FUNCTION FC 23 : VOID
TITLE = Bock for actuating several cycled valves
//Erstellung:
//Datum       Bearbeiter                                                   Version
//--------------------------------------------------------------------------------
//14.06.99    A.Kirchgessner(kia)                                         01.00.00
//
//Änderungen:
//Nr. Datum    Bearb Änderung                                       Marke  Version
//--------------------------------------------------------------------------------
//01  16.07.99 kia   Fehlerbeseitigung                                    01.00.01
//02  12.08.99 sra   Fehlerbeseitigung mit Parameteränderung              01.01.00
//03  19.10.99 sra   Anpassung an neue Struktur                           01.02.00
//04  10.07.00 sra   Fehlerbeseitigung Taktgenerierung                    01.02.01
//05  10.07.00 sra   Änderung in Eingangsparameter                        01.03.00
//06  19.09.00 sra   komplette Überarbeitung / neue Struktur              02.00.00
//07  18.01.01 gea   Erweiterung auf 10 Ventile / neue Struktur           02.01.00
//08  27.03.02 sra   Meldung "Ventil in Betrieb" auch im Handmode   (008) 02.01.01
//09  04.02.03 kal   Fehlerbeseitigung Dauertakt                    (009) 02.01.02
//10  31.10.05 sra   Ansteuerung Handbedienung im Automode rücksetz.
//                   Handbedienung zentral sperren                  (010) 02.02.00
//11  18.02.09 kmj   Objektststatus für OP ergänzt                  (011) 02.03.00
//12  20.03.09 kal   Objektststatus für OP ergänzt (überarbeitet)   (012) 02.03.01
//13  24.04.09 gea   Handmode zurücksetzen wenn Handmode gesperrt   (013) 02.03.02
//14  05.12.13 sra   "Anlage ein" eingefügt (Not-Aus-Konzept)       (014) 02.04.00
//15  14.11.14 bhl   Anzeige "#io_Ventil_in_Betrieb" im Handmode    (015) 02.04.01
//16  11.08.15 sra   "#io_Ventil_in_Betrieb" nur wenn "Anlage ein"  (016) 02.04.02
//________________________________________________________________________________
//Eingesetzte Bausteine:
//
//FC2 : Version 01.01.XX
//________________________________________________________________________________
//Funktion:
//
//Der Baustein taktet die einzelnen Ventile der Reihe nach durch (Anzahl der 
//Ventile max. 10 Stück). 
//
//Die Ausgänge werden nur angesteuert wenn der Eingang "in_Anlage_ein" = true
//ist. Diese Funktion ist vorhanden, um bei einem Not-Halt die Anlage vor 
//unkontrolliertem Einschalten zu schützen. 
//
//Im Handmode werden die ausgewählten Ventile dauerhaft angesteuert. 
//
AUTHOR : kia
FAMILY : AZO
VERSION : 0.0
VAR_INPUT
  in_Handbedienung_erlaubt : BOOL ;	//1 = manual operation permitted, 0 = manual operation not permitted/locked
  in_Anlage_ein : BOOL ;	//Anlage bzw. Anlagenbereich nach Not-Halt freigegeben
  in_Ansteuerung_Ventil_T1 : BOOL ;	//Actuation of valve position 1 in automatic mode with cycle 1
  in_Ansteuerung_Ventil_T2 : BOOL ;	//Actuation of valve position 1 in automatic mode with cycle 2
END_VAR
VAR_IN_OUT
  io_Ausgang_Ventil_1 : BOOL ;	//Output 1. Valve
  io_Ausgang_Ventil_2 : BOOL ;	//Output 2. Valve
  io_Ausgang_Ventil_3 : BOOL ;	//Output 3. Valve
  io_Ausgang_Ventil_4 : BOOL ;	//Output 4. Valve
  io_Ausgang_Ventil_5 : BOOL ;	//Output 5. Valve
  io_Ausgang_Ventil_6 : BOOL ;	//Output 6. Valve
  io_Ausgang_Ventil_7 : BOOL ;	//Output 7. Valve
  io_Ausgang_Ventil_8 : BOOL ;	//Output 8. Valve
  io_Ausgang_Ventil_9 : BOOL ;	//Output 9. Valve
  io_Ausgang_Ventil_10 : BOOL ;	//Output 10. Valve
  io_Ventil_in_Betrieb : BOOL ;	//Signal "valve in operation" (actuated)
  io_Ventilstruktur : ANY ;	//ANY pointer of valve structure
END_VAR
VAR_TEMP
  Ventilansteuerung : BOOL ;	//Freigabe ein Ventil anzusteuern
  Freigabe_Takt : BOOL ;	//Cycle enable
  Rueckmeldung : BOOL ;	//wenn eines der Ventil agesteuert ist --> 1-Signal
  Start_mit_Impuls : BOOL ;
  Taktanzahl_erreicht : BOOL ;
  Dauertakt : BOOL ;	//Continuous cycle
  positive_Flanke : BOOL ;
  Hilfs_Anzahl_Takte : INT ;	//Sollvorgabe für FC2
  Aktuelles_Ventil : INT ;	//aktuelles Ventil
  Hilfswort_1 : INT ;
  Impulszeit_Takt : REAL ;
  Pausezeit_Takt : REAL ;
  Zeitzaehler : REAL ;
  Taktzaehler : INT ;
  Objektstatus : INT ;
END_VAR
BEGIN
NETWORK
TITLE = Anfangs-DW der Struktur aus ANY-Zeiger auslesen
      L     P##io_Ventilstruktur;
      LAR2;
      L     D [AR2,P#6.0];
      LAR2;	//Pointer auf Structuranfang
NETWORK
TITLE = Umschaltung Hand-/Automatikmode 
      A     DIX [AR2,P#3.6];	// Handmode von Farbgrafik (Struktur)
      AN    DIX [AR2,P#5.1];	// Handmode gesperrt (Struktur)
      AN    M 0.0;	// Handbedienung zentral sperren (010)
      S     DIX [AR2,P#3.5];	// Handmode zu Farbgrafik (Struktur)
      ON    DIX [AR2,P#3.6];	// Handmode von Farbgrafik (Struktur)
      ON    #in_Handbedienung_erlaubt;
      O     M 0.0;	// Handbedienung zentral sperren (010)
      O     DIX [AR2,P#5.1];	// Handmode gesperrt (Struktur) (013)
      R     DIX [AR2,P#3.5];	// Handmode zu Farbgrafik (Struktur)
      R     DIX [AR2,P#3.6];	// Handmode von Farbgrafik (Struktur) (010)
NETWORK
TITLE = Ansteuerung Handmode zurücksetzen
//(010) 
      AN    DIX [AR2,P#3.5];	// Handmode zu Farbgrafik (Struktur)
      R     DIX [AR2,P#3.7];	// Ansteuerung des 1. Ventils im Handmode von Farbgrafik (Struktur)
      R     DIX [AR2,P#4.0];	// Ansteuerung des 2. Ventils im Handmode von Farbgrafik (Struktur)
      R     DIX [AR2,P#4.1];	// Ansteuerung des 3. Ventils im Handmode von Farbgrafik (Struktur)
      R     DIX [AR2,P#4.2];	// Ansteuerung des 4. Ventils im Handmode von Farbgrafik (Struktur)
      R     DIX [AR2,P#4.3];	// Ansteuerung des 5. Ventils im Handmode von Farbgrafik (Struktur)
      R     DIX [AR2,P#4.4];	// Ansteuerung des 6. Ventils im Handmode von Farbgrafik (Struktur)
      R     DIX [AR2,P#4.5];	// Ansteuerung des 7. Ventils im Handmode von Farbgrafik (Struktur)
      R     DIX [AR2,P#4.6];	// Ansteuerung des 8. Ventils im Handmode von Farbgrafik (Struktur)
      R     DIX [AR2,P#4.7];	// Ansteuerung des 9. Ventils im Handmode von Farbgrafik (Struktur)
      R     DIX [AR2,P#5.0];	// Ansteuerung des 10. Ventils im Handmode von Farbgrafik (Struktur)
NETWORK
TITLE = Rueckmeldung Ventile + Ventilansteuerung
      O     #io_Ausgang_Ventil_1;
      O     #io_Ausgang_Ventil_2;
      O     #io_Ausgang_Ventil_3;
      O     #io_Ausgang_Ventil_4;
      O     #io_Ausgang_Ventil_5;
      O     #io_Ausgang_Ventil_6;
      O     #io_Ausgang_Ventil_7;
      O     #io_Ausgang_Ventil_8;
      O     #io_Ausgang_Ventil_9;
      O     #io_Ausgang_Ventil_10;
      =     #Rueckmeldung;
      =     #Ventilansteuerung;
NETWORK
TITLE = Daten für Takt in temporäre Variablen laden
//(009) komplettes Netzwerk gelöscht.
//Dauertakt nur, wenn Bit in Struktur = TRUE 
//Anzahl Takte ist egal!!!
      A     DIX [AR2,P#5.2];	// Start mit Impuls (Struktur)
      =     #Start_mit_Impuls;
      A     DIX [AR2,P#5.3];	// Taktanzahl erreicht (Struktur)
      =     #Taktanzahl_erreicht;
      A     DIX [AR2,P#5.4];	// Dauertakt (Struktur)
      =     #Dauertakt;
      L     DID [AR2,P#22.0];	// Impuls-/Pausezähler (Struktur)
      T     #Zeitzaehler;
      L     DIW [AR2,P#28.0];	// Taktzähler (Struktur)
      T     #Taktzaehler;
NETWORK
TITLE = Sollanzahl Takte
      AN    #Dauertakt;
      JC    ST_1;
      L     DIW [AR2,P#30.0];	// Anzahl Ventile (Struktur)
      T     #Hilfs_Anzahl_Takte;
ST_1: NOP   0;
      A     #Dauertakt;
      JC    ST_2;
      L     DIW [AR2,P#26.0];	// Sollanzahl Takte (Struktur)
      T     #Hilfs_Anzahl_Takte;
ST_2: NOP   0;
NETWORK
TITLE = Freigabe Takt
      A     #in_Anlage_ein;	// (014)
      A(;	// (014)
      O     #in_Ansteuerung_Ventil_T1;
      O     #in_Ansteuerung_Ventil_T2;
      );	// (014)
      =     #Freigabe_Takt;
NETWORK
TITLE = Takt umkopieren
      L     DID [AR2,P#6.0];	// Impulszeit Befüllung (Struktur)
      T     #Impulszeit_Takt;
      L     DID [AR2,P#10.0];	// Pausezeit Befüllung (Struktur)
      T     #Pausezeit_Takt;
      A     #in_Ansteuerung_Ventil_T1;
      JC    E_Tk;
      L     DID [AR2,P#14.0];	// Impulszeit Entleerung (Struktur)
      T     #Impulszeit_Takt;
      L     DID [AR2,P#18.0];	// Pausezeit Entleerung (Struktur)
      T     #Pausezeit_Takt;
E_Tk: NOP   0;
NETWORK
TITLE = Takt generieren
      CALL  FC 2 (
           in_Freigabe              := #Freigabe_Takt,
           in_Rueckmeldung          := #Rueckmeldung,
           in_Start_mit_Impuls      := #Start_mit_Impuls,
           in_Dauertakt             := #Dauertakt,
           in_Impuls                := M 1.7,
           in_Impulszeit_in_100ms   := MW 6,
           in_Impulszeit            := #Impulszeit_Takt,
           in_Pausezeit             := #Pausezeit_Takt,
           in_Sollanzahl_Takte      := #Hilfs_Anzahl_Takte,
           io_Taktausgang           := #Ventilansteuerung,
           io_Taktanzahl_erreicht   := #Taktanzahl_erreicht,
           io_Zeitzaehler           := #Zeitzaehler,
           io_Taktzaehler           := #Taktzaehler);
NETWORK
TITLE = aktuelles Ventil
      L     #Taktzaehler;
      L     DIW [AR2,P#30.0];	// Anzahl Ventile (Struktur)
      /I;
      T     #Hilfswort_1;
      L     #Hilfswort_1;
      L     DIW [AR2,P#30.0];	// Anzahl Ventile (Struktur)
      *I;
      L     -1;
      *I;
      L     #Taktzaehler;
      +I;
      L     1;
      +I;
      T     #Aktuelles_Ventil;
NETWORK
TITLE = aktuelles Ventil prüfen
      A(;
      L     #Aktuelles_Ventil;
      L     1;
      >=I;
      );
      A(;
      L     #Aktuelles_Ventil;
      L     DIW [AR2,P#30.0];	// Anzahl Ventile (Struktur)
      <=I;
      );
      JC    M1;
      L     1;
      T     #Aktuelles_Ventil;
M1:   NOP   0;
NETWORK
TITLE = Ansteuerung Ventil 1
      A     #in_Anlage_ein;	// (014)
      A(;	// (014)
      A(;
      L     #Aktuelles_Ventil;
      L     1;
      ==I;
      );
      A(;	// Automatikmode
      AN    DIX [AR2,P#3.5];	// Handmode zu Farbgrafik (Struktur)
      A     #Ventilansteuerung;
      AN    #Taktanzahl_erreicht;
      );
      O;	// Handmode 
      A     DIX [AR2,P#3.5];	// Handmode zu Farbgrafik (Struktur)
      A     DIX [AR2,P#3.7];	// Ansteuerung des 1. Ventils im Handmode von Farbgrafik (Struktur)
      );	// (014)
      =     #io_Ausgang_Ventil_1;
NETWORK
TITLE = Ansteuerung Ventil 2
      A     #in_Anlage_ein;	// (014)
      A(;	// (014)
      A(;
      L     #Aktuelles_Ventil;
      L     2;
      ==I;
      );
      A(;	// Automatikmode
      AN    DIX [AR2,P#3.5];	// Handmode zu Farbgrafik (Struktur)
      A     #Ventilansteuerung;
      AN    #Taktanzahl_erreicht;
      );
      O;	// Handmode 
      A     DIX [AR2,P#3.5];	// Handmode zu Farbgrafik (Struktur)
      A     DIX [AR2,P#4.0];	// Ansteuerung des 2. Ventils im Handmode von Farbgrafik (Struktur)
      );	// (014)
      =     #io_Ausgang_Ventil_2;
NETWORK
TITLE = Ansteuerung Ventil 3
      A     #in_Anlage_ein;	// (014)
      A(;	// (014)
      A(;
      L     #Aktuelles_Ventil;
      L     3;
      ==I;
      );
      A(;	// Automatikmode
      AN    DIX [AR2,P#3.5];	// Handmode zu Farbgrafik (Struktur)
      A     #Ventilansteuerung;
      AN    #Taktanzahl_erreicht;
      );
      O;	// Handmode 
      A     DIX [AR2,P#3.5];	// Handmode zu Farbgrafik (Struktur)
      A     DIX [AR2,P#4.1];	// Ansteuerung des 3. Ventils im Handmode von Farbgrafik (Struktur)
      );	// (014)
      =     #io_Ausgang_Ventil_3;
NETWORK
TITLE = Ansteuerung Ventil 4
      A     #in_Anlage_ein;	// (014)
      A(;	// (014)
      A(;
      L     #Aktuelles_Ventil;
      L     4;
      ==I;
      );
      A(;	// Automatikmode
      AN    DIX [AR2,P#3.5];	// Handmode zu Farbgrafik (Struktur)
      A     #Ventilansteuerung;
      AN    #Taktanzahl_erreicht;
      );
      O;	// Handmode 
      A     DIX [AR2,P#3.5];	// Handmode zu Farbgrafik (Struktur)
      A     DIX [AR2,P#4.2];	// Ansteuerung des 4. Ventils im Handmode von Farbgrafik (Struktur)
      );	// (014)
      =     #io_Ausgang_Ventil_4;
NETWORK
TITLE = Ansteuerung Ventil 5
      A     #in_Anlage_ein;	// (014)
      A(;	// (014)
      A(;
      L     #Aktuelles_Ventil;
      L     5;
      ==I;
      );
      A(;	// Automatikmode
      AN    DIX [AR2,P#3.5];	// Handmode zu Farbgrafik (Struktur)
      A     #Ventilansteuerung;
      AN    #Taktanzahl_erreicht;
      );
      O;	// Handmode 
      A     DIX [AR2,P#3.5];	// Handmode zu Farbgrafik (Struktur)
      A     DIX [AR2,P#4.3];	// Ansteuerung des 5. Ventils im Handmode von Farbgrafik (Struktur)
      );	// (014)
      =     #io_Ausgang_Ventil_5;
NETWORK
TITLE = Ansteuerung Ventil 6
      A     #in_Anlage_ein;	// (014)
      A(;	// (014)
      A(;
      L     #Aktuelles_Ventil;
      L     6;
      ==I;
      );
      A(;	// Automatikmode
      AN    DIX [AR2,P#3.5];	// Handmode zu Farbgrafik (Struktur)
      A     #Ventilansteuerung;
      AN    #Taktanzahl_erreicht;
      );
      O;	// Handmode 
      A     DIX [AR2,P#3.5];	// Handmode zu Farbgrafik (Struktur)
      A     DIX [AR2,P#4.4];	// Ansteuerung des 6. Ventils im Handmode von Farbgrafik (Struktur)
      );	// (014)
      =     #io_Ausgang_Ventil_6;
NETWORK
TITLE = Ansteuerung Ventil 7
      A     #in_Anlage_ein;	// (014)
      A(;	// (014)
      A(;
      L     #Aktuelles_Ventil;
      L     7;
      ==I;
      );
      A(;	// Automatikmode
      AN    DIX [AR2,P#3.5];	// Handmode zu Farbgrafik (Struktur)
      A     #Ventilansteuerung;
      AN    #Taktanzahl_erreicht;
      );
      O;	// Handmode 
      A     DIX [AR2,P#3.5];	// Handmode zu Farbgrafik (Struktur)
      A     DIX [AR2,P#4.5];	// Ansteuerung des 7. Ventils im Handmode von Farbgrafik (Struktur)
      );	// (014)
      =     #io_Ausgang_Ventil_7;
NETWORK
TITLE = Ansteuerung Ventil 8
      A     #in_Anlage_ein;	// (014)
      A(;	// (014)
      A(;
      L     #Aktuelles_Ventil;
      L     8;
      ==I;
      );
      A(;	// Automatikmode
      AN    DIX [AR2,P#3.5];	// Handmode zu Farbgrafik (Struktur)
      A     #Ventilansteuerung;
      AN    #Taktanzahl_erreicht;
      );
      O;	// Handmode 
      A     DIX [AR2,P#3.5];	// Handmode zu Farbgrafik (Struktur)
      A     DIX [AR2,P#4.6];	// Ansteuerung des 8. Ventils im Handmode von Farbgrafik (Struktur)
      );	// (014)
      =     #io_Ausgang_Ventil_8;
NETWORK
TITLE = Ansteuerung Ventil 9
      A     #in_Anlage_ein;	// (014)
      A(;	// (014)
      A(;
      L     #Aktuelles_Ventil;
      L     9;
      ==I;
      );
      A(;	// Automatikmode
      AN    DIX [AR2,P#3.5];	// Handmode zu Farbgrafik (Struktur)
      A     #Ventilansteuerung;
      AN    #Taktanzahl_erreicht;
      );
      O;	// Handmode 
      A     DIX [AR2,P#3.5];	// Handmode zu Farbgrafik (Struktur)
      A     DIX [AR2,P#4.7];	// Ansteuerung des 9. Ventils im Handmode von Farbgrafik (Struktur)
      );	// (014)
      =     #io_Ausgang_Ventil_9;
NETWORK
TITLE = Ansteuerung Ventil 10
      A     #in_Anlage_ein;	// (014)
      A(;	// (014)
      A(;
      L     #Aktuelles_Ventil;
      L     10;
      ==I;
      );
      A(;	// Automatikmode
      AN    DIX [AR2,P#3.5];	// Handmode zu Farbgrafik (Struktur)
      A     #Ventilansteuerung;
      AN    #Taktanzahl_erreicht;
      );
      O;	// Handmode 
      A     DIX [AR2,P#3.5];	// Handmode zu Farbgrafik (Struktur)
      A     DIX [AR2,P#5.0];	// Ansteuerung des 10. Ventils im Handmode von Farbgrafik (Struktur)
      );	// (014)
      =     #io_Ausgang_Ventil_10;
NETWORK
TITLE = Ausgang Betrieb
      AN    DIX [AR2,P#3.5];	// (015) Handmode zu Farbgrafik (Struktur)
      A     #in_Anlage_ein;	// (016)
      A(;
      O     #in_Ansteuerung_Ventil_T1;
      O     #in_Ansteuerung_Ventil_T2;	// (008)
      );
      A     #Dauertakt;
      O;
      AN    DIX [AR2,P#3.5];	// (015) Handmode zu Farbgrafik (Struktur)
      A     #in_Anlage_ein;	// (016)
      A(;
      O     #in_Ansteuerung_Ventil_T1;
      O     #in_Ansteuerung_Ventil_T2;
      );
      AN    #Dauertakt;
      AN    #Taktanzahl_erreicht;
      O;
      A     DIX [AR2,P#3.5];	// Handmode zu Farbgrafik (Struktur)
      A     #in_Anlage_ein;	// (016)
      A(;
      O     #io_Ausgang_Ventil_1;	// (008)
      O     #io_Ausgang_Ventil_2;	// (008)
      O     #io_Ausgang_Ventil_3;	// (008)
      O     #io_Ausgang_Ventil_4;	// (008)
      O     #io_Ausgang_Ventil_5;	// (008)
      O     #io_Ausgang_Ventil_6;	// (008)
      O     #io_Ausgang_Ventil_7;	// (008)
      O     #io_Ausgang_Ventil_8;	// (008)
      O     #io_Ausgang_Ventil_9;	// (008)
      O     #io_Ausgang_Ventil_10;	// (008)
      );
      =     #io_Ventil_in_Betrieb;
NETWORK
TITLE = Flankenauswertung Ausgang Ventil für Schalthäufigkeitzähler
//Es wird die Schalthäufigkeit der Ventile gezählt !  
      O     #io_Ausgang_Ventil_1;
      O     #io_Ausgang_Ventil_2;
      O     #io_Ausgang_Ventil_3;
      O     #io_Ausgang_Ventil_4;
      O     #io_Ausgang_Ventil_5;
      O     #io_Ausgang_Ventil_6;
      O     #io_Ausgang_Ventil_7;
      O     #io_Ausgang_Ventil_8;
      O     #io_Ausgang_Ventil_9;
      O     #io_Ausgang_Ventil_10;
      FP    DIX [AR2,P#32.3];	// Flankenmerker Ausgang (Struktur)
      =     #positive_Flanke;
NETWORK
TITLE = Schalthäufigkeitzähler
      ON    DIX [AR2,P#0.3];	// Kennung Schalthäufigkeitzähler ein (Struktur)
      ON    #positive_Flanke;
      JC    ESHZ;
      L     1.000000e+00;
      L     DID [AR2,P#34.0];	// Schalthäufigkeitzähler (Struktur)
      +R;
      T     DID [AR2,P#34.0];	// Schalthäufigkeitzähler (Struktur)
ESHZ: NOP   0;
NETWORK
TITLE = Schalthäufigkeitzähler zurücksetzten
      AN    DIX [AR2,P#32.0];	// Reset Schalthäufigkeitzähler (Struktur)
      JC    E_RS;
      L     0.000000e+00;
      T     DID [AR2,P#34.0];	// Schalthäufigkeitzähler (Struktur)
      CLR;
      =     DIX [AR2,P#32.0];	// Reset Schalthäufigkeitzähler (Struktur)
E_RS: NOP   0;
NETWORK
TITLE = Warnmeldung Schalthäufigkeitzähler erzeugen
      A(;
      L     DID [AR2,P#34.0];	// Schalthäufigkeitzähler (Struktur)
      L     DID [AR2,P#38.0];	// Sollwert Warnung (Struktur)
      >R;
      );
      A(;
      L     DID [AR2,P#38.0];	// Sollwert Warnung (Struktur)
      L     0.000000e+00;
      <>R;
      );
      =     DIX [AR2,P#32.1];	// Warnmeldung Schalthäufigkeitzähler (Struktur)
NETWORK
TITLE = Alarmmeldung Schalthäufigkeitzähler erzeugen
      A(;
      L     DID [AR2,P#34.0];	// Schalthäufigkeitzähler (Struktur)
      L     DID [AR2,P#42.0];	// Sollwert Alarm (Struktur)
      >R;
      );
      A(;
      L     DID [AR2,P#42.0];	// Sollwert Alarm (Struktur)
      L     0.000000e+00;
      <>R;
      );
      =     DIX [AR2,P#32.2];	// Warnmeldung Schalthäufigkeitzähler (Struktur)
NETWORK
TITLE = Objektstatus für Visualisation OP (011)(012)
//Stati:
//-------
//1 = kein Ventil angesteuert ==> Farbvorschlag weiß
//5 = ein ventil in Betrieb ==> Farbvorschlag grün
//
// 1 = nicht in Betrieb, keine Störung ==> Farbvorschlag grau
      L     1;
      AN    #io_Ventil_in_Betrieb;
      JC    disp;
// 5 = angesteuert, nicht in Betrieb, keine Störung ==> Farbvorschlag grün
      L     5;
      A     #io_Ventil_in_Betrieb;
      JC    disp;
      L     0;
disp: T     #Objektstatus;
NETWORK
TITLE = Daten in Struktur speichern
      A     #in_Anlage_ein;	// (014)
      =     DIX [AR2,P#5.5];	// (014) Anlage ein (Struktur)
      A     #io_Ausgang_Ventil_1;
      =     DIX [AR2,P#2.0];	// Ausgang Ventil 1 (Struktur)
      A     #io_Ausgang_Ventil_2;
      =     DIX [AR2,P#2.1];	// Ausgang Ventil 2 (Struktur)
      A     #io_Ausgang_Ventil_3;
      =     DIX [AR2,P#2.2];	// Ausgang Ventil 3 (Struktur)
      A     #io_Ausgang_Ventil_4;
      =     DIX [AR2,P#2.3];	// Ausgang Ventil 4 (Struktur)
      A     #io_Ausgang_Ventil_5;
      =     DIX [AR2,P#2.4];	// Ausgang Ventil 5 (Struktur)
      A     #io_Ausgang_Ventil_6;
      =     DIX [AR2,P#2.5];	// Ausgang Ventil 6 (Struktur)
      A     #io_Ausgang_Ventil_7;
      =     DIX [AR2,P#2.6];	// Ausgang Ventil 7 (Struktur)
      A     #io_Ausgang_Ventil_8;
      =     DIX [AR2,P#2.7];	// Ausgang Ventil 8 (Struktur)
      A     #io_Ausgang_Ventil_9;
      =     DIX [AR2,P#3.0];	// Ausgang Ventil 9 (Struktur)
      A     #io_Ausgang_Ventil_10;
      =     DIX [AR2,P#3.1];	// Ausgang Ventil 10 (Struktur)
      A     #io_Ventil_in_Betrieb;
      =     DIX [AR2,P#3.4];	// Ventil in Betrieb (Struktur)
      A     #Taktanzahl_erreicht;
      =     DIX [AR2,P#5.3];	// Taktanzahl erreicht (Struktur)
      L     #Zeitzaehler;
      T     DID [AR2,P#22.0];	// Impuls-/Pausezähler (Struktur)
      L     #Taktzaehler;
      T     DIW [AR2,P#28.0];	// Taktzähler (Struktur)
      L     #Objektstatus;	// (011)
      T     DIW [AR2,P#48.0];	// #Objektstatus  (Struktur)   // (011)
END_FUNCTION

FUNCTION FC 24 : VOID
TITLE = Block for debouncing and fault monitoring of a binary input
//Building:
//Date         Editor                                                     Version
//--------------------------------------------------------------------------------
//22.09.99     (jm)                                                       01.00.00
//
//Modifications:
//No. Date     Edit  Description                                    Index Version
//--------------------------------------------------------------------------------
//01  29.09.00 sra   komplette Überarbeitung / neue Struktur        ()    02.00.00
//02  16.06.05 sra   Änderung INC 1 -> + 1                         (002)  02.00.01
//03  04.09.06 sra   Änderung Störungsquittierung                  (003)  02.01.00
//04  08.07.10 jm    Störzeit 0 möglich                            (004)  02.01.01
//05  06.06.16 kal/sra komplette Überarbeitung (wie TIA-Portal)     ()    03.00.00
//06  12.06.16 sra   Änderung Signal "Eingang verarbeitet"         (006)  03.01.00
//07  13.12.17 gea   Objektstatus betätig/störung (neu)            (007)  03.02.00
//                   Objektstatus nicht betätig/störung (neu)
//                   Eingang verarbeitet bei Störung ausgeben
//08  26.01.18 gea   Objektstatus Fehlerbeseitigung                (008)  03.02.01
//
//________________________________________________________________________________
//Functional description:
//
//The Binary Input Object includes the following functions
//- The input can be turned (0 = input is active) -> configuration value
//- Depending on the Parameter "in_fault_state", it is possible to select whether
//  log. 0 or log. 1 will represent the fault.
//- The input signal can be debounced in both directions with a seperate time
//  -> Real values in structure
//- The input signal can be counted -> value in structure -> configuration value
//
//The main application for the function are level indicators.
//
AUTHOR : jm
VERSION : 3.2
VAR_INPUT
  in_Handbedienung_erlaubt : BOOL ;
  in_Anlage_ein : BOOL ;
  in_Eingang : BOOL ;
  in_Eingang_drehen : BOOL ;
  in_Eingang_entprellen : BOOL ;
  in_Stoerauswertung_aktiv : BOOL ;
  in_Quitt_Stoerung_noetig : BOOL ;
  in_Stoer_Zustand : BOOL ;
  in_Quitt_Stoerung : BOOL ;
END_VAR
VAR_IN_OUT
  io_Eingang_verarbeitet : BOOL ;
  io_Stoerung : BOOL ;
  io_Struktur : ANY ;
END_VAR
VAR_TEMP
  Eingang_nach_Drehung : BOOL ;
  Eingang_nach_Entprellung : BOOL ;
  Diskrepanz : BOOL ;
  Freigabe_Entprellung_HIG : BOOL ;
  Ausgang_Entprellung_HIGH : BOOL ;
  Freigabe_Entprellung_LOW : BOOL ;
  Ausgang_Entprellung_LOW : BOOL ;
  positive_Flanke : BOOL ;
  Objektstatus : INT ;
  Temp_DB : INT ;
  Sollzeit_Entprellung_HIG : REAL ;
  Istzeit_Entprellung_HIGH : REAL ;
  Sollzeit_Entprellung_LOW : REAL ;
  Istzeit_entprellung_LOW : REAL ;
END_VAR
BEGIN
NETWORK
TITLE = Anfangs-DW der Struktur aus ANY-Zeiger auslesen
      L     P##io_Struktur;
      LAR2;
      L     D [AR2,P#6.0];
      LAR2;
NETWORK
TITLE = Daten aus Struktur lesen
      A     DIX [AR2,P#3.4];
      =     #Eingang_nach_Drehung;
      A     DIX [AR2,P#3.5];
      =     #Eingang_nach_Entprellung;
      A     DIX [AR2,P#3.6];
      =     #Ausgang_Entprellung_HIGH;
      A     DIX [AR2,P#3.7];
      =     #Ausgang_Entprellung_LOW;
      L     DID [AR2,P#8.0];
      T     #Sollzeit_Entprellung_HIG;
      L     DID [AR2,P#12.0];
      T     #Istzeit_Entprellung_HIGH;
      L     DID [AR2,P#16.0];
      T     #Sollzeit_Entprellung_LOW;
      L     DID [AR2,P#20.0];
      T     #Istzeit_entprellung_LOW;
NETWORK
TITLE = Eingang ggf. drehen
      A     #in_Eingang;
      AN    #in_Eingang_drehen;
      O;
      AN    #in_Eingang;
      A     #in_Eingang_drehen;
      =     #Eingang_nach_Drehung;
NETWORK
TITLE = Umschaltung Hand-/Automatikmode 
      A     DIX [AR2,P#2.7];	// Handmode von Farbgrafik (Struktur)
      AN    DIX [AR2,P#3.1];	// Handmode gesperrt (Struktur)
      AN    M 0.0;	// Handbedienung zentral sperren 
      S     DIX [AR2,P#2.6];	// Handmode zu Farbgrafik (Struktur)
      ON    DIX [AR2,P#2.7];	// Handmode von Farbgrafik (Struktur)
      ON    #in_Handbedienung_erlaubt;
      O     M 0.0;	// Handbedienung zentral sperren 
      O     DIX [AR2,P#3.1];	// Handmode gesperrt (Struktur)
      R     DIX [AR2,P#2.6];	// Handmode zu Farbgrafik (Struktur)
      R     DIX [AR2,P#2.7];	// Handmode von Farbgrafik (Struktur)
NETWORK
TITLE = Handzustand im Automatikmode speichern
      AN    DIX [AR2,P#2.6];	// Handmode zu Farbgrafik (Struktur)
      JCN   SAM;
      A     #Eingang_nach_Drehung;
      AN    #in_Eingang_drehen;
      =     DIX [AR2,P#3.0];	// Zustand Handmode (Struktur)
      AN    #Eingang_nach_Drehung;
      A     #in_Eingang_drehen;
      =     DIX [AR2,P#3.0];	// Zustand Handmode (Struktur)
SAM:  NOP   0;
NETWORK
TITLE = Zustand nach Drehung im Handmode überschreiben
      A     DIX [AR2,P#2.6];	// Handmode zu Farbgrafik (Struktur)
      JCN   SHM;
      A     DIX [AR2,P#3.0];	// Zustand Handmode (Struktur)
      =     #Eingang_nach_Drehung;
SHM:  NOP   0;
NETWORK
TITLE = Diskrepanz feststellen
// Automode
      AN    DIX [AR2,P#2.6];	// Handmode zu Farbgrafik (Struktur)
      A     #in_Stoerauswertung_aktiv;
      AN    #in_Eingang;	//Störung = log. 0
      AN    #in_Stoer_Zustand;
      O;
      AN    DIX [AR2,P#2.6];	// Handmode zu Farbgrafik (Struktur)
      A     #in_Stoerauswertung_aktiv;
      A     #in_Eingang;	//Störung = log. 1
      A     #in_Stoer_Zustand;
      O;
// Handmode 
      A     DIX [AR2,P#2.6];	// Handmode zu Farbgrafik (Struktur)
      A     #in_Stoerauswertung_aktiv;
      AN    #Eingang_nach_Drehung;	//Störung = log. 0
      AN    #in_Stoer_Zustand;
      O;
      A     DIX [AR2,P#2.6];	// Handmode zu Farbgrafik (Struktur)
      A     #in_Stoerauswertung_aktiv;
      A     #Eingang_nach_Drehung;	//Störung = log. 1
      A     #in_Stoer_Zustand;
      =     #Diskrepanz;
NETWORK
TITLE = Stoerungszaehler
      A     #in_Quitt_Stoerung_noetig;
      AN    #in_Quitt_Stoerung;
      A     #io_Stoerung;
      O;
      A     #Diskrepanz;
      AN    #in_Quitt_Stoerung;
      O;
      AN    #in_Quitt_Stoerung_noetig;
      A     #Diskrepanz;
      JC    SZ1;
      L     0;	// Wenn keine Diskrepanz dann Zähler löschen
      T     DIW [AR2,P#6.0];	// Istzeit Störung (Struktur)
      JU    ESZ;
// Störungszähler in jeder Sekunde erhöhen
SZ1:  O     #io_Stoerung;
      ON    M 4.5;	// Sekundenimpuls (Standardmerker)
      JC    ESZ;
      L     DIW [AR2,P#6.0];	// Istzeit Störung (Struktur)
      +     1;	// (002)
      T     DIW [AR2,P#6.0];	// Istzeit Störung (Struktur)
ESZ:  NOP   0;
NETWORK
TITLE = Störmeldung ausgeben
      L     DIW [AR2,P#6.0];	// Istzeit Störung (Struktur)
      L     DIW [AR2,P#4.0];	// Sollzeit Störung (Struktur)
      >I;
      =     #io_Stoerung;
NETWORK
TITLE = Stoerung quittieren
      O     #Diskrepanz;	// Stoerung steht noch an
      ON    #io_Stoerung;
      JC    ESQ;
      ON    #in_Quitt_Stoerung_noetig;	// Stoerung muß quittiert werden ?
      JC    SQ1;	// Stoerung muß nicht quittiert werden
      A     #in_Quitt_Stoerung;
SQ1:  R     #io_Stoerung;
ESQ:  NOP   0;
NETWORK
TITLE = Entprellung HIGH
      A     #Eingang_nach_Drehung;
      A     #in_Eingang_entprellen;
      =     #Freigabe_Entprellung_HIG;
      CALL  FC 3 (
           in_Freigabe              := #Freigabe_Entprellung_HIG,
           in_Reset                 := M 0.3,
           in_Impuls                := M 1.7,
           in_Impulszeit_in_100ms   := MW 6,
           in_Verzoegerungsart      := B#16#45,
           in_Verzoegerungszeit     := #Sollzeit_Entprellung_HIG,
           io_Ausgangssignal        := #Ausgang_Entprellung_HIGH,
           io_Zeitzaehler           := #Istzeit_Entprellung_HIGH);
NETWORK
TITLE = Entprellung LOW
      AN    #Eingang_nach_Drehung;
      A     #in_Eingang_entprellen;
      =     #Freigabe_Entprellung_LOW;
      CALL  FC 3 (
           in_Freigabe              := #Freigabe_Entprellung_LOW,
           in_Reset                 := M 0.3,
           in_Impuls                := M 1.7,
           in_Impulszeit_in_100ms   := MW 6,
           in_Verzoegerungsart      := B#16#45,
           in_Verzoegerungszeit     := #Sollzeit_Entprellung_LOW,
           io_Ausgangssignal        := #Ausgang_Entprellung_LOW,
           io_Zeitzaehler           := #Istzeit_entprellung_LOW);
NETWORK
TITLE = Entprellung
      A     #Eingang_nach_Drehung;
      A     #in_Eingang_entprellen;
      A     #Ausgang_Entprellung_HIGH;
      S     #Eingang_nach_Entprellung;
      AN    #Eingang_nach_Drehung;
      A     #in_Eingang_entprellen;
      A     #Ausgang_Entprellung_LOW;
      R     #Eingang_nach_Entprellung;
      NOP   0;
NETWORK
TITLE = verarbeitetes Eingangssignal zuweisen
// Automatikmode
      AN    DIX [AR2,P#2.6];	// Handmode zu Farbgrafik (Struktur)
      AN    #in_Eingang_entprellen;
      A     #Eingang_nach_Drehung;
//      UN    #io_Stoerung                // (006) (007)
      O;
// Automatikmode
      AN    DIX [AR2,P#2.6];	// Handmode zu Farbgrafik (Struktur)
      A     #in_Eingang_entprellen;
      A     #Eingang_nach_Entprellung;
//      UN    #io_Stoerung                // (006) (007)
      O;
// Handmode 
      A     DIX [AR2,P#2.6];	// Handmode zu Farbgrafik (Struktur)
      A     DIX [AR2,P#3.0];	// Zustand Handmode (Struktur)
      AN    #in_Eingang_drehen;
//      UN    #io_Stoerung                // (006) (007)
      O;
// Handmode 
      A     DIX [AR2,P#2.6];	// Handmode zu Farbgrafik (Struktur)
      AN    DIX [AR2,P#3.0];	// Zustand Handmode (Struktur)
      A     #in_Eingang_drehen;
//      UN    #io_Stoerung                // (006) (007)
      =     #io_Eingang_verarbeitet;
NETWORK
TITLE = Flankenauswertung Ausgang Ventil für Schalthäufigkeitzähler
      A     #io_Eingang_verarbeitet;
      FP    DIX [AR2,P#24.3];	// Flankenmerker Ausgang (Struktur)
      =     #positive_Flanke;
NETWORK
TITLE = Schalthäufigkeitzähler
      ON    DIX [AR2,P#0.3];	// Kennung Schalthäufigkeitzähler ein (Struktur)
      ON    #positive_Flanke;
      JC    ESHZ;
      L     1.000000e+00;
      L     DID [AR2,P#26.0];	// Schalthäufigkeitzähler (Struktur)
      +R;
      T     DID [AR2,P#26.0];	// Schalthäufigkeitzähler (Struktur)
ESHZ: NOP   0;
NETWORK
TITLE = Schalthäufigkeitzähler zurücksetzten
      AN    DIX [AR2,P#24.0];	// Reset Schalthäufigkeitzähler (Struktur)
      JC    E_RS;
      L     0.000000e+00;
      T     DID [AR2,P#26.0];	// Schalthäufigkeitzähler (Struktur)
      CLR;
      =     DIX [AR2,P#24.0];	// Reset Schalthäufigkeitzähler (Struktur)
E_RS: NOP   0;
NETWORK
TITLE = Warnmeldung Schalthäufigkeitszähler erzeugen
      A(;
      L     DID [AR2,P#26.0];	// Schalthäufigkeitzähler (Struktur)
      L     DID [AR2,P#30.0];	// Sollwert Warnung (Struktur)
      >R;
      );
      A(;
      L     DID [AR2,P#30.0];	// Sollwert Warnung (Struktur)
      L     0.000000e+00;
      <>R;
      );
      =     DIX [AR2,P#24.1];	// Warnmeldung Schalthäufigkeitzähler (Struktur)
NETWORK
TITLE = Alarmmeldung Schalthäufigkeitszähler erzeugen
      A(;
      L     DID [AR2,P#26.0];	// Schalthäufigkeitzähler (Struktur)
      L     DID [AR2,P#34.0];	// Sollwert Alarm (Struktur)
      >R;
      );
      A(;
      L     DID [AR2,P#34.0];	// Sollwert Alarm (Struktur)
      L     0.000000e+00;
      <>R;
      );
      =     DIX [AR2,P#24.2];	// Alarmmeldung Schalthäufigkeitzähler (Struktur)
NETWORK
TITLE =  Objektstatus für Visualisation OP (009) (010)
// 19 = Anlage nicht ein (interlock) ==> Farbvorschlag orange
      L     19;
      AN    #in_Anlage_ein;
      AN    #io_Stoerung;
      JC    disp;
// 1 = nicht betaetigt ==> Farbvorschlag weiß
      L     1;
      AN    #io_Eingang_verarbeitet;
      AN    #io_Stoerung;
      AN    DIX [AR2,P#1.0];	// Kennung "invers"
      O;
      A     #io_Eingang_verarbeitet;
      AN    #io_Stoerung;
      A     DIX [AR2,P#1.0];	// Kennung "invers"
      JC    disp;
// 5 = betätigt ==> Farbvorschlag grün(gelb)
      L     5;
      A     #io_Eingang_verarbeitet;
      AN    #io_Stoerung;
      AN    DIX [AR2,P#1.0];	// Kennung "invers"
      O;
      AN    #io_Eingang_verarbeitet;
      AN    #io_Stoerung;
      A     DIX [AR2,P#1.0];	// Kennung "invers"
      JC    disp;
// 14 = Störung, nicht betätigt, Störung ==> Farbvorschlag rot/weiß
      L     14;	// (007)
      AN    #io_Eingang_verarbeitet;	// (007)
      A     #io_Stoerung;	// (007)
      AN    DIX [AR2,P#1.0];	// (007) Kennung "invers"
      A     #in_Anlage_ein;	// (007)
      O;	// (007)
      A     #io_Eingang_verarbeitet;	// (007)
      A     #io_Stoerung;	// (007)
      A     DIX [AR2,P#1.0];	// (007) Kennung "invers"
      A     #in_Anlage_ein;	// (007)
      JC    disp;	// (007)
// 15 = Störung, nicht betätigtt, Störung ==> Farbvorschlag rot/grün(gelb)
      L     15;	// (008)
      A     #io_Eingang_verarbeitet;	// (007)
      A     #io_Stoerung;	// (007)
      AN    DIX [AR2,P#1.0];	// (007) Kennung "invers"
      A     #in_Anlage_ein;	// (007)
      O;	// (007)
      AN    #io_Eingang_verarbeitet;	// (007)
      A     #io_Stoerung;	// (007) (008)
      A     DIX [AR2,P#1.0];	// (007) Kennung "invers"
      A     #in_Anlage_ein;	// (007)
      JC    disp;	// (007)
// 16 = Störung
      L     16;
      A     #io_Stoerung;
      JC    disp;
      L     0;
disp: T     #Objektstatus;
NETWORK
TITLE = Daten in Struktur kopieren
      A     #io_Eingang_verarbeitet;
      =     DIX [AR2,P#2.0];	// Eingang verarbeitet (Struktur)
      A     #in_Eingang;
      =     DIX [AR2,P#2.1];	// Eingang (Struktur)
      A     #in_Eingang_drehen;
      =     DIX [AR2,P#2.2];	// Eingang drehen (Struktur)
      A     #in_Eingang_entprellen;
      =     DIX [AR2,P#2.3];	// Eingang entprellen (Struktur)
      A     #in_Stoer_Zustand;
      =     DIX [AR2,P#2.4];	// Störzustand (Struktur)
      A     #io_Stoerung;
      =     DIX [AR2,P#2.5];	// Störung (Struktur)
      A     #in_Anlage_ein;	// (006)
      =     DIX [AR2,P#3.2];	// (006) Anlage ein (Struktur) 
      A     #Eingang_nach_Drehung;
      =     DIX [AR2,P#3.4];
      A     #Eingang_nach_Entprellung;
      =     DIX [AR2,P#3.5];
      A     #Ausgang_Entprellung_HIGH;
      =     DIX [AR2,P#3.6];
      A     #Ausgang_Entprellung_LOW;
      =     DIX [AR2,P#3.7];
      AN    #Ausgang_Entprellung_HIGH;
      JCN   noHi;
      L     #Istzeit_Entprellung_HIGH;
      T     DID [AR2,P#12.0];
noHi: NOP   0;
      AN    #Ausgang_Entprellung_LOW;
      JCN   noLo;
      L     #Istzeit_entprellung_LOW;
      T     DID [AR2,P#20.0];
noLo: NOP   0;
      L     #Objektstatus;
      T     DIW [AR2,P#48.0];	// #Objektstatus  (Struktur) 
END_FUNCTION

FUNCTION FC 25 : VOID
TITLE = Lamp Functiomnality - copied from TIA Library
NAME : standard
VERSION : 0.1
VAR_INPUT
  Steady : BOOL ;
  Flash : BOOL ;
  DoubleFlash : BOOL ;
  LampTest : BOOL ;
END_VAR
VAR_OUTPUT
  Lamp : BOOL ;
END_VAR
BEGIN
NETWORK
TITLE = Lamp Operation
      A     #Steady;
      AN    #Flash;
      AN    #DoubleFlash;
      AN    M 1.5;
      O;
      A     #Flash;
      AN    #DoubleFlash;
      A     M 2.4;
      AN    M 1.5;
      O;
      A     #DoubleFlash;
      A     M 2.4;
      A     M 2.1;
      AN    M 1.5;
      O;
      A     M 1.5;
      O;
      A     #LampTest;
      =     #Lamp;
END_FUNCTION

FUNCTION FC 28 : VOID
TITLE = Block for analog input
//Building:
//Date         Editor                                                     Version
//--------------------------------------------------------------------------------
//06.03.2017   (gea)                                                      01.00.00
//
//Modifications:
//No. Date     Edit  Description                                    Index Version
//--------------------------------------------------------------------------------
//01a 20.06.17 gea   Filter implemented                             (001) 01.01.00
//01b 17.01.18 gea   no configuration clean-up to allow dynamic     (001b)
//                   alarm enable
//________________________________________________________________________________
//Functional description:
//
//The analog Input Object includes the following functions
//- 
//
AUTHOR : gea
VERSION : 1.1
VAR_INPUT
  ManOpEn : BOOL ;	// Enable Manual mode
  ManModeTrack : BOOL ;	// Manual mode PV tracking
  OVErrEn : BOOL ;	// overflow/underflow/broken wire error enable
  AlarmHiEn : BOOL ;	// Alarm high enable
  AlarmHiAckEn : BOOL ;	// Alarm high acknowledge enable
  AlarmLoEn : BOOL ;	//Alarm low enable
  AlarmLoAckEn : BOOL ;	//Alarm low acknowledge enable
  SwitchEn : BOOL ;	//Switch enable
  SwitchPol : BOOL ;	//Switch polarity
  DigitMin : INT ;	// scaling digit max
  DigitMax : INT ;	// scaling digit min
  ValueMin : REAL ;	// scaling value max
  ValueMax : REAL ;	// scaling value min
  ValueSubs : REAL ;	// substitude value
  Filter : REAL ;	//filter value = 1.0 ...
  Configuration : WORD ;	// external Configuration (0=use internal)
  UOM : INT ;	// external Uom  (0=use internal)
  iSystemOn : BOOL ;	// System activated
  iwDigit : INT ;	// input digit value
  aAlarmHiAck : BOOL ;	// Alarm high acknowledge
  aAlarmLoAck : BOOL ;	//Alarm low acknowledge
END_VAR
VAR_IN_OUT
  PVAct : REAL ;
  Switch : BOOL ;
  fAlarmHi : BOOL ;
  fAlarmLo : BOOL ;
  fScalingErr : BOOL ;
  fOVErr : BOOL ;
  ioStructure : ANY ;
END_VAR
VAR_TEMP
  State : INT ;
  tempReal1 : REAL ;
  tempReal2 : REAL ;
  tempDB : INT ;
  PVIn : REAL ;
END_VAR
BEGIN
NETWORK
TITLE =  get start byte of structure
      L     P##ioStructure;
      LAR2;
      L     W [AR2,P#4.0];
      T     #tempDB;
      OPN   DI [#tempDB];
      L     D [AR2,P#6.0];
      LAR2;
NETWORK
TITLE =  external  configuration
      L     #Configuration;
      L     0;
      ==I;
      JC    NECO;
      L     #Configuration;
      L     0;
      <>I;
      =     DIX [AR2,P#0.0];	// AnalogInOn on
      L     #Configuration;
      L     2#1000;
      AW;
      L     0;
      <>I;
      =     DIX [AR2,P#0.3];	// switch counter on
      L     #Configuration;
      L     2#10000;
      AW;
      L     0;
      <>I;
      =     DIX [AR2,P#0.4];	// switch level input
      L     #Configuration;
      L     2#100000;
      AW;
      L     0;
      <>I;
      =     DIX [AR2,P#0.5];	// switch level hysteresis input
      L     #Configuration;
      L     2#100000000;
      AW;
      L     0;
      <>I;
      =     DIX [AR2,P#1.0];	// alarm high level input
      L     #Configuration;
      L     2#1000000000;
      AW;
      L     0;
      <>I;
      =     DIX [AR2,P#1.1];	// alarm low level input
      L     #Configuration;
      L     2#10000000000;
      AW;
      L     0;
      <>I;
      =     DIX [AR2,P#1.2];	// alarm level hysteresis input
NECO: NOP   0;
      L     #UOM;
      L     0;
      ==I;
      JC    NEUO;
      L     #UOM;
      T     DIW [AR2,P#2.0];
NEUO: NOP   0;
NETWORK
TITLE =  clean up configuration
//      UN    #SwitchEn                                                                     //(001b)
//      R     DIX [AR2,P#0.4]             // switch level input                             //(001b)
//      R     DIX [AR2,P#0.5]             // switch level hysteresis input                  //(001b)
//      R     DIX [AR2,P#0.3]             // switch counter on                              //(001b)
//      UN    #AlarmHiEn                                                                    //(001b)
//      R     DIX [AR2,P#1.0]             // alarm high level input                         //(001b)
//      UN    #AlarmLoEn                                                                    //(001b)
//      R     DIX [AR2,P#1.1]             // alarm low level input                          //(001b)
//      UN    #AlarmHiEn                                                                    //(001b)
//      UN    #AlarmLoEn                                                                    //(001b)
//      R     DIX [AR2,P#1.2]             // alarm level hysteresis input                   //(001b)
NETWORK
TITLE =  selection manual mode
      A     DIX [AR2,P#4.1];	// ManModeOp
      AN    DIX [AR2,P#4.2];	// ManModeLock
      AN    M 0.0;	// manual mode general disabled
      S     DIX [AR2,P#4.0];	// ManModAct
      ON    DIX [AR2,P#4.1];	// ManModeOp
      ON    #ManOpEn;	// manual mode local disabled
      O     M 0.0;	// manual mode general disabled
      O     DIX [AR2,P#4.2];	// ManModeLock
      R     DIX [AR2,P#4.0];	// ManModAct
      R     DIX [AR2,P#4.1];	// ManModeOp
NETWORK
TITLE =  overflow / underflow / broken wire check
      O(;
      L     #iwDigit;
      L     32511;
      >I;
      );	//overflow
      O(;
      A(;
      L     #iwDigit;
      L     -32512;
      <I;
      );
      A(;
      L     #DigitMin;
      L     0;
      <>I;	//bipolar
      );
      );	//underflow bipolar
      O(;
      A(;
      L     #iwDigit;
      L     -4864;
      <I;
      );
      A(;
      L     #DigitMin;
      L     0;
      ==I;	//unipolar
      );
      );	//underflow //unipolar
      A     #OVErrEn;	//enable overflow / underflow error
      =     #fOVErr;
NETWORK
TITLE =  scaling of PV
//Val = ValueMin + (ValueMax-ValueMin)*(iwDigit-DigitMin)/(DigitMax-DigitMin)
// (network holds code this reader does not know; not shown)
NETWORK
TITLE =  substidue PV
      O     #fScalingErr;
      O     #fOVErr;
      AN    DIX [AR2,P#4.0];	// ManModAct
      JCN   PVSU;
      L     #ValueSubs;
      T     #PVIn;	//(001)
PVSU: NOP   0;
NETWORK
TITLE = manual mode PV
      A     DIX [AR2,P#4.0];	// ManModAct
      JCN   PVMA;
      L     DID [AR2,P#10.0];	//ManModePV      
      T     #PVIn;	//(001)
PVMA: NOP   0;
NETWORK
TITLE = Filter PV
//(001) 
// 
      L     1.000000e+00;
      L     #Filter;
      <R;
      JC    FIOK;
      L     #PVIn;	//in case the number of counts is 0 or negative
      JU    FNOK;
FIOK: L     1.000000e+00;
      -R;
      L     #PVAct;
      *R;
      L     #PVIn;
      +R;
      L     #Filter;
      /R;
FNOK: T     #PVAct;
NETWORK
TITLE =  track manual mode value in automatic
      AN    DIX [AR2,P#4.0];	// ManModAct
      A     #ManModeTrack;
      JCN   PVTK;
      L     #PVAct;
      T     DID [AR2,P#10.0];	//ManModePV      
PVTK: NOP   0;
NETWORK
TITLE = Alarm high
      A(;
      L     #PVAct;
      L     DID [AR2,P#14.0];	//AlarmHiPV
      >R;	//PVact>AlarmHiPV
      );
      A     #AlarmHiEn;
      S     #fAlarmHi;
      A(;
      L     DID [AR2,P#14.0];	//AlarmHiPV
      L     DID [AR2,P#22.0];	//AlarmHystPV
      -R;
      L     #PVAct;
      TAK;
      <R;	//PVact<(AlarmHiPV-AlarmHystPV
      );
      A(;
      A     #AlarmHiAckEn;
      A     #aAlarmHiAck;
      ON    #AlarmHiAckEn;
      );
      ON    #AlarmHiEn;
      ON    #iSystemOn;
      R     #fAlarmHi;
NETWORK
TITLE = Alarm low
      A(;
      L     #PVAct;
      L     DID [AR2,P#18.0];	//AlarmLoPV
      <R;	//PVact<AlarmLoPV
      );
      A     #AlarmLoEn;
      S     #fAlarmLo;
      A(;
      L     DID [AR2,P#18.0];	//AlarmLoPV
      L     DID [AR2,P#22.0];	//AlarmHystPV
      +R;
      L     #PVAct;
      TAK;
      >R;	//PVact<(AlarmHiPV-AlarmHystPV
      );
      A(;
      A     #AlarmLoAckEn;
      A     #aAlarmLoAck;
      ON    #AlarmLoAckEn;
      );
      ON    #AlarmLoEn;
      ON    #iSystemOn;
      R     #fAlarmLo;
NETWORK
TITLE = switch
      L     DID [AR2,P#26.0];	//SwitchLevelPV
      L     DID [AR2,P#30.0];	//SwitchHysteresis
      -R;
      T     #tempReal1;	//Switch level high hysteresis
      L     DID [AR2,P#26.0];	//SwitchLevelPV
      L     DID [AR2,P#30.0];	//SwitchHysteresis
      +R;
      T     #tempReal2;	//Switch level low hysteresis
      A     #SwitchEn;
      A     #SwitchPol;
      A(;
      L     #PVAct;
      L     DID [AR2,P#26.0];	//SwitchLevelPV
      >R;
      );	//(SwitchPolarity=positive) * (PVAct>SwitchLevel)
      O;
      A     #SwitchEn;
      AN    #SwitchPol;
      A(;
      L     #PVAct;
      L     DID [AR2,P#26.0];	//SwitchLevelPV
      <R;
      );	//(SwitchPolarity=negative) * (PVAct<SwitchLevel)
      S     #Switch;
      A     #SwitchEn;
      A     #SwitchPol;
      A(;
      L     #PVAct;
      L     #tempReal1;	//Switch level high hysteresis
      <R;
      );	//(SwitchPolarity=positive) * (PVAct<(SwitchLevel-SwitchLevelhysteresis)
      O;
      A     #SwitchEn;
      AN    #SwitchPol;
      A(;
      L     #PVAct;
      L     #tempReal2;	//Switch level low hysteresis
      >R;
      );	//(SwitchPolarity=negative) * (PVAct<(SwitchLevel+SwitchLevelhysteresis)
      ON    #SwitchEn;
      R     #Switch;
NETWORK
TITLE =  Switch counter count up
      A     #Switch;
      FP    DIX [AR2,P#34.3];	// Switch counter edge
      A     DIX [AR2,P#0.3];	// Configuarion switching counter
      JCN   SCUP;
      L     1.000000e+00;
      L     DID [AR2,P#36.0];	// Switch counter
      +R;
      T     DID [AR2,P#36.0];	// Switch counter
SCUP: NOP   0;
NETWORK
TITLE =  Switch counter reset
      A     DIX [AR2,P#34.0];	// Switch counter Reset
      JCN   SCRE;
      R     DIX [AR2,P#34.0];	// Switch counter Reset
      L     0.000000e+00;
      T     DID [AR2,P#36.0];	// Switch counter
SCRE: NOP   0;
NETWORK
TITLE = Switch counter warning
      A(;
      L     DID [AR2,P#36.0];	// Switch counter
      L     DID [AR2,P#40.0];	// Switch counter warning count
      >R;
      );
      A(;
      L     DID [AR2,P#40.0];	// Switch counter warning count
      L     0.000000e+00;
      <>R;
      );
      =     DIX [AR2,P#34.1];	// Switch counter warning 
NETWORK
TITLE = Switch counter alarm
      A(;
      L     DID [AR2,P#36.0];	// Switch counter
      L     DID [AR2,P#44.0];	// Switch counter alarm count
      >R;
      );
      A(;
      L     DID [AR2,P#44.0];	// Sollwert Alarm (Struktur)
      L     0.000000e+00;
      <>R;
      );
      =     DIX [AR2,P#34.2];	// Switch counter alarm 
NETWORK
TITLE =  Objektstatus für Visualisation OP (009) (010)
// 9 = scaling/overflow/underflow/broken wire: substitude value ==> grey 
      L     9;
      O     #fScalingErr;
      O     #fOVErr;
      JC    disp;
// 19 = system not on (interlock) ==> orange
      L     19;
      AN    #iSystemOn;
      JC    disp;
// 16 = alarm high ==> red
      L     16;
      O     #fAlarmHi;
      JC    disp;
// 16 = alarm low ==> yellow
      L     13;
      O     #fAlarmLo;
      JC    disp;
// 5 = switch on ==> green
      L     5;
      A     #Switch;
      A     #SwitchEn;
      JC    disp;
// 1 = switch off ==> white
      L     1;
      AN    #Switch;
      A     #SwitchEn;
      JC    disp;
      L     0;
disp: T     #State;
NETWORK
TITLE =  save data to structure
      A     #iSystemOn;
      =     DIX [AR2,P#4.3];
      A     #fScalingErr;
      =     DIX [AR2,P#4.4];
      A     #fOVErr;
      =     DIX [AR2,P#4.5];
      A     #fAlarmHi;
      =     DIX [AR2,P#4.6];
      A     #AlarmHiEn;
      =     DIX [AR2,P#4.7];
      A     #aAlarmHiAck;
      =     DIX [AR2,P#5.0];
      A     #fAlarmLo;
      =     DIX [AR2,P#5.1];
      A     #AlarmLoEn;
      =     DIX [AR2,P#5.2];
      A     #aAlarmLoAck;
      =     DIX [AR2,P#5.3];
      L     #PVAct;
      T     DID [AR2,P#6.0];
      A     #Switch;
      =     DIX [AR2,P#5.4];
      A     #SwitchEn;
      =     DIX [AR2,P#5.5];
      L     #State;
      T     DIW [AR2,P#48.0];	// #Objektstatus  (Struktur) 
END_FUNCTION

FUNCTION FC 29 : VOID
TITLE = Block for pressure analog input
//Building:
//Date         Editor                                                     Version
//--------------------------------------------------------------------------------
//10.05.2017   (gea)                                                      01.00.00
//
//Modifications:
//No. Date     Edit  Description                                    Index Version
//--------------------------------------------------------------------------------
//01  
//________________________________________________________________________________
//Functional description:
//
//The Pressure Analogue Input Object includes the following functions
//- Check of overflow with substitude value
//- scaling of input value
//- check of pressure levels
//- mode selection 
//  manual mode (empty / convey / overpressure | zero pint adjustment)
//- overpressure detection (with delay)
//- overpressure alarm (with delay)
//- empty pressure detection (with delay)
//- active pressure detection 
//- adjustment of zeropoint (autoamtic / manual)
//- data structure for HMI connection
//
AUTHOR : gea
VERSION : 1.0
VAR_INPUT
  ManOpEn : BOOL ;	// Enable Manual mode
  ManModeTrack : BOOL ;	// Manual mode PV tracking
  NegEvalEn : BOOL ;	// overpressure=0; underpressure=1
  OVErrEn : BOOL ;	// overflow/underflow/broken wire error enable
  AlarmOprEn : BOOL ;	// Alarm high enable
  AlarmOprAckEn : BOOL ;	// Alarm high acknowledge enable
  DigitMin : INT ;	// scaling digit max
  DigitMax : INT ;	// scaling digit min
  ValueMin : REAL ;	// scaling value max
  ValueMax : REAL ;	// scaling value min
  ValueSubs : REAL ;	// substitude value
  Configuration : WORD ;	// external Configuration (0=use internal)
  UOM : INT ;	// external Uom  (0=use internal)
  iSystemOn : BOOL ;	// System activated
  iwDigit : INT ;	// input digit value
  iActive : BOOL ;	// Pressure montioring active
  aAlarmOprAck : BOOL ;	// Alarm high acknowledge
END_VAR
VAR_IN_OUT
  PVAct : REAL ;
  fAlarmOpr : BOOL ;
  OverPressure : BOOL ;
  EmptyPressure : BOOL ;
  ActivePressure : BOOL ;
  fScalingErr : BOOL ;
  fOVErr : BOOL ;
  fParErr : BOOL ;
  ioStructure : ANY ;
END_VAR
VAR_TEMP
  State : INT ;
  tempReal1 : REAL ;
  tempReal2 : REAL ;
  tempDB : INT ;
  PVActRaw : REAL ;
  ScaleingErrPV : BOOL ;
  ScaleingErrOffset : BOOL ;
END_VAR
BEGIN
NETWORK
TITLE =  get start byte of structure
      L     P##ioStructure;
      LAR2;
      L     W [AR2,P#4.0];
      T     #tempDB;
      OPN   DI [#tempDB];
      L     D [AR2,P#6.0];
      LAR2;
NETWORK
TITLE =  external  configuration
      L     #Configuration;
      L     0;
      ==I;
      JC    NECO;
      L     #Configuration;
      L     0;
      <>I;
      =     DIX [AR2,P#0.0];	// PressureAinOn
      L     #Configuration;
      L     2#1000;
      AW;
      L     0;
      <>I;
      =     DIX [AR2,P#0.3];	// counter overpressure on
      L     #Configuration;
      L     2#10000;
      AW;
      L     0;
      <>I;
      =     DIX [AR2,P#0.4];	// counter emptypressure on
      L     #Configuration;
      L     2#100000;
      AW;
      L     0;
      <>I;
      =     DIX [AR2,P#0.5];	// counter activepressure on
      L     #Configuration;
      L     2#100000000;
      AW;
      L     0;
      <>I;
      =     DIX [AR2,P#1.0];	// overpressure parameter on
      L     #Configuration;
      L     2#1000000000;
      AW;
      L     0;
      <>I;
      =     DIX [AR2,P#1.1];	// emptypressure parameter on
      L     #Configuration;
      L     2#10000000000;
      AW;
      L     0;
      <>I;
      =     DIX [AR2,P#1.2];	// activeypressure parameter on
      L     #Configuration;
      L     2#1000000000000;
      AW;
      L     0;
      <>I;
      =     DIX [AR2,P#1.4];	// manual operation simulation on
      L     #Configuration;
      L     2#10000000000000;
      AW;
      L     0;
      <>I;
      =     DIX [AR2,P#1.5];	// manual operation adjust on
NECO: NOP   0;
      L     #UOM;
      L     0;
      ==I;
      JC    NEUO;
      L     #UOM;
      T     DIW [AR2,P#2.0];
NEUO: NOP   0;
NETWORK
TITLE =  clean up configuration
      O     DIX [AR2,P#0.3];	// counter overpressure on
      R     DIX [AR2,P#0.4];	// counter emptypressure on
      O     DIX [AR2,P#0.3];	// counter overpressure on
      O     DIX [AR2,P#0.4];	// counter emptypressure on
      R     DIX [AR2,P#0.5];	// counter activepressure on
NETWORK
TITLE =  selection manual mode
      A     DIX [AR2,P#4.1];	// ManModeOp
      AN    DIX [AR2,P#4.2];	// ManModeLock
      AN    M 0.0;	// manual mode general disabled
      S     DIX [AR2,P#4.0];	// ManModAct
      ON    DIX [AR2,P#4.1];	// ManModeOp
      ON    #ManOpEn;	// manual mode local disabled
      O     M 0.0;	// manual mode general disabled
      O     DIX [AR2,P#4.2];	// ManModeLock
      R     DIX [AR2,P#4.0];	// ManModAct
      R     DIX [AR2,P#4.1];	// ManModeOp
NETWORK
TITLE =  overflow / underflow / broken wire check
      O(;
      L     #iwDigit;
      L     32511;
      >I;
      );	//overflow
      O(;
      A(;
      L     #iwDigit;
      L     -32512;
      <I;
      );
      A(;
      L     #DigitMin;
      L     0;
      <>I;	//bipolar
      );
      );	//underflow bipolar
      O(;
      A(;
      L     #iwDigit;
      L     -4864;
      <I;
      );
      A(;
      L     #DigitMin;
      L     0;
      ==I;	//unipolar
      );
      );	//underflow //unipolar
      A     #OVErrEn;	//enable overflow / underflow error
      =     #fOVErr;
NETWORK
TITLE =  scaling of PV
//Val = ValueMin + (ValueMax-ValueMin)*(iwDigit-DigitMin)/(DigitMax-DigitMin)
// (network holds code this reader does not know; not shown)
NETWORK
TITLE =  substidue PV
      O     #fScalingErr;
      O     #fOVErr;
      AN    DIX [AR2,P#4.0];	// ManModAct
      JCN   PVSU;
      L     #ValueSubs;
      T     #PVAct;
PVSU: NOP   0;
NETWORK
TITLE =  manual mode PV: off
      A     DIX [AR2,P#4.0];	// ManModAct
      AN    DIX [AR2,P#4.3];	// ManOpPressureEmpty
      AN    DIX [AR2,P#4.4];	// ManOpPressureConveying
      AN    DIX [AR2,P#4.5];	// ManOpPressureAlarm
      A     DIX [AR2,P#1.4];	// ManOpSimEn
      JCN   PVMO;
      L     0.000000e+00;
      T     #PVAct;
PVMO: NOP   0;
NETWORK
TITLE =  manual mode PV: Emptypressure
      A     DIX [AR2,P#4.0];	// ManModAct
      A     DIX [AR2,P#4.3];	// ManOpPressureEmpty
      AN    DIX [AR2,P#4.4];	// ManOpPressureConveying
      AN    DIX [AR2,P#4.5];	// ManOpPressureAlarm
      A     DIX [AR2,P#1.4];	// ManOpSimEn
      JCN   PVME;
      L     DID [AR2,P#24.0];	//EmptypressurePV     
      L     DID [AR2,P#28.0];	//ActivePressurePV    
      -R;
      L     2.000000e+00;
      /R;
      L     DID [AR2,P#28.0];	//ActivePressurePV    
      +R;
      T     #PVAct;
PVME: NOP   0;
NETWORK
TITLE =  manual mode PV: convey pressure
      A     DIX [AR2,P#4.0];	// ManModAct
      A     DIX [AR2,P#4.4];	// ManOpPressureConveying
      AN    DIX [AR2,P#4.5];	// ManOpPressureAlarm
      A     DIX [AR2,P#1.4];	// ManOpSimEn
      JCN   PVMC;
      L     DID [AR2,P#16.0];	//MaxpressurePV     
      L     DID [AR2,P#24.0];	//EmptypressurePV     
      -R;
      L     2.000000e+00;
      /R;
      L     DID [AR2,P#24.0];	//EmptypressurePV     
      +R;
      T     #PVAct;
PVMC: NOP   0;
NETWORK
TITLE =  manual mode PV: overpressure
      A     DIX [AR2,P#4.0];	// ManModAct
      A     DIX [AR2,P#4.5];	// ManOpPressureAlarm
      A     DIX [AR2,P#1.4];	// ManOpSimEn
      JCN   PVMA;
      L     DID [AR2,P#16.0];	//MaxpressurePV     
      T     #PVAct;
PVMA: NOP   0;
NETWORK
TITLE =  check Parameter
// (network holds code this reader does not know; not shown)
NETWORK
TITLE =  overpressure detection
      A(;
      L     #PVAct;
      L     DID [AR2,P#16.0];	//MaxpressurePV     
      >=R;
      );
      AN    #NegEvalEn;
      A     #iActive;
      O;
      A(;
      L     #PVAct;
      L     DID [AR2,P#16.0];	//MaxpressurePV     
      <=R;
      );
      A     #NegEvalEn;
      A     #iActive;
      S     #OverPressure;
      A(;
      L     #PVAct;
      L     DID [AR2,P#20.0];	//MinpressurePV 
      <=R;
      );
      AN    #NegEvalEn;
      O;
      A(;
      L     #PVAct;
      L     DID [AR2,P#20.0];	//MinpressurePV 
      >=R;
      );
      A     #NegEvalEn;
      ON    #iActive;
      R     #OverPressure;
NETWORK
TITLE =  emptypressure detection
      A(;
      L     #PVAct;
      L     DID [AR2,P#24.0];	//EmptypressurePV     
      <=R;
      );
      AN    #NegEvalEn;
      A     #iActive;
      O;
      A(;
      L     #PVAct;
      L     DID [AR2,P#24.0];	//EmptypressurePV     
      >=R;
      );
      A     #NegEvalEn;
      A     #iActive;
      JCN   EPDC;
      A     M 4.5;
      AN    #EmptyPressure;
      L     DIW [AR2,P#38.0];	// EmptyDelayCounter
      JCN   EPDR;
      +     1;
      JU    EPDR;
EPDC: L     0;
EPDR: T     DIW [AR2,P#38.0];	// EmptyDelayCounter
      L     DIW [AR2,P#32.0];	// EmptyDelay
      >=I;
      =     #EmptyPressure;
NETWORK
TITLE =  activepressure detection
      A(;
      L     #PVAct;
      L     DID [AR2,P#28.0];	//ActivePressurePV    
      >=R;
      );
      A     #iActive;
      AN    #NegEvalEn;
      O;
      A(;
      L     #PVAct;
      L     DID [AR2,P#28.0];	//ActivePressurePV    
      <=R;
      );
      A     #iActive;
      A     #NegEvalEn;
      JCN   APDC;
      A     M 4.5;
      AN    #ActivePressure;
      L     DIW [AR2,P#40.0];	// ActiveDelayCounter
      JCN   APDR;
      +     1;
      JU    APDR;
APDC: L     0;
APDR: T     DIW [AR2,P#40.0];	// ActiveDelayCounter
      L     DIW [AR2,P#34.0];	// ActiveDelay
      >=I;
      =     #ActivePressure;
NETWORK
TITLE =  Alarm overpressure
      A     #OverPressure;
      A     #AlarmOprEn;
      A     #iActive;
      JCN   OPDC;
      A     M 4.5;
      AN    #fAlarmOpr;
      L     DIW [AR2,P#42.0];	// AlarmDelayCounter
      JCN   OPDR;
      +     1;
      JU    OPDR;
OPDC: L     0;
OPDR: T     DIW [AR2,P#42.0];	// AlarmDelayCounter
      L     DIW [AR2,P#36.0];	// AlarmDelay
      >=I;
      S     #fAlarmOpr;
      AN    #OverPressure;
      A(;
      A     #AlarmOprAckEn;
      A     #aAlarmOprAck;
      ON    #AlarmOprAckEn;
      );
      ON    #AlarmOprEn;
      ON    #iSystemOn;
      ON    #iActive;
      R     #fAlarmOpr;
NETWORK
TITLE =  adjust automatic
// (network holds code this reader does not know; not shown)
NETWORK
TITLE =  adjust manual
      AN    DIX [AR2,P#4.0];	// ManModeAct
      A     DIX [AR2,P#1.5];	// parameter.MapOpAdjustEn
      A     DIX [AR2,P#4.6];	// ManOpPressureAdjust
      =     DIX [AR2,P#6.4];	// ManAdjustReq
      A     DIX [AR2,P#1.5];	// parameter.MapOpAdjustEn
      A     DIX [AR2,P#4.6];	// ManOpPressureAdjust
      AN    #iActive;
      A     DIX [AR2,P#6.4];	// ManAdjustReq
      A     DIX [AR2,P#6.5];	// ManAdjustRdy
      JCN   ADMA;
      L     #PVActRaw;
      T     DID [AR2,P#12.0];	//PressureOffset
      SET;	// done!
      R     DIX [AR2,P#4.6];	// ManOpPressureAdjust
ADMA: NOP   0;
      ON    DIX [AR2,P#1.5];	// parameter.MapOpAdjustEn
      R     DIX [AR2,P#4.6];	// ManOpPressureAdjust
NETWORK
TITLE =  Switch counter count up
      A     #OverPressure;
      A     DIX [AR2,P#0.3];	// parameter.counterOverPressure
      O;
      A     #EmptyPressure;
      A     DIX [AR2,P#0.4];	// parameter.counterEmptyPressure
      O;
      A     #ActivePressure;
      A     DIX [AR2,P#0.5];	// parameter.counterActivePressure
      FP    DIX [AR2,P#6.7];	// Switch counter edge
      JCN   SCUP;
      L     1.000000e+00;
      L     DID [AR2,P#44.0];	// Switch counter
      +R;
      T     DID [AR2,P#44.0];	// Switch counter
SCUP: NOP   0;
NETWORK
TITLE =  Switch counter reset
      A     DIX [AR2,P#6.6];	// Switch counter Reset
      O;
      AN    DIX [AR2,P#0.3];	// parameter.counterOverPressure
      AN    DIX [AR2,P#0.5];	// parameter.counterEmptyPressure
      AN    DIX [AR2,P#0.4];	// parameter.counterActivePressure
      JCN   SCRE;
      R     DIX [AR2,P#6.6];	// Switch counter Reset
      L     0.000000e+00;
      T     DID [AR2,P#44.0];	// Switch counter
SCRE: NOP   0;
NETWORK
TITLE =  track manual mode value in automatic
      AN    DIX [AR2,P#4.0];	// ManModAct
      A     #ManModeTrack;
      AN    #fParErr;
      JCN   PVTK;
      AN    #ActivePressure;
      AN    #EmptyPressure;
      AN    #OverPressure;
      R     DIX [AR2,P#4.3];	// ManOpPressureEmpty
      R     DIX [AR2,P#4.4];	// ManOpPressureConveying
      R     DIX [AR2,P#4.5];	// ManOpPressureAlarm
      A     #ActivePressure;
      A     #EmptyPressure;
      AN    #OverPressure;
      S     DIX [AR2,P#4.3];	// ManOpPressureEmpty
      R     DIX [AR2,P#4.4];	// ManOpPressureConveying
      R     DIX [AR2,P#4.5];	// ManOpPressureAlarm
      A     #ActivePressure;
      AN    #EmptyPressure;
      AN    #OverPressure;
      R     DIX [AR2,P#4.3];	// ManOpPressureEmpty
      S     DIX [AR2,P#4.4];	// ManOpPressureConveying
      R     DIX [AR2,P#4.5];	// ManOpPressureAlarm
      A     #ActivePressure;
      AN    #EmptyPressure;
      A     #OverPressure;
      R     DIX [AR2,P#4.3];	// ManOpPressureEmpty
      R     DIX [AR2,P#4.4];	// ManOpPressureConveying
      S     DIX [AR2,P#4.5];	// ManOpPressureAlarm
PVTK: NOP   0;
NETWORK
TITLE =  Objektstatus für Visualisation OP (009) (010)
// 9 = scaling/overflow/underflow/broken wire: substitude value ==> grey 
      L     9;
      O     #fScalingErr;
      O     #fOVErr;
      JC    disp;
// 19 = system not on (interlock) ==> orange
      L     19;
      AN    #iSystemOn;
      JC    disp;
// 16 = alarm overpressure ==> red
      L     16;
      A     #fAlarmOpr;
      JC    disp;
// 16 = overpressure ==> yellow
      L     13;
      A     #OverPressure;
      AN    #fAlarmOpr;
      JC    disp;
// 5 = switch on ==> green
      L     5;
      A     #ActivePressure;
      AN    #EmptyPressure;
      JC    disp;
// 1 = switch off ==> cyan
      L     1;
      A     #ActivePressure;
      A     #EmptyPressure;
      JC    disp;
      L     0;
disp: T     #State;
NETWORK
TITLE =  save data to structure
      A     #iSystemOn;
      =     DIX [AR2,P#4.7];
      A     #fScalingErr;
      =     DIX [AR2,P#5.0];
      A     #fOVErr;
      =     DIX [AR2,P#5.1];
      A     #fParErr;
      =     DIX [AR2,P#5.2];
      A     #fAlarmOpr;
      =     DIX [AR2,P#5.3];
      A     #AlarmOprEn;
      =     DIX [AR2,P#5.4];
      A     #aAlarmOprAck;
      =     DIX [AR2,P#5.5];
      A     #OverPressure;
      =     DIX [AR2,P#5.6];
      A     #EmptyPressure;
      =     DIX [AR2,P#5.7];
      A     #ActivePressure;
      =     DIX [AR2,P#6.0];
      A     #iActive;
      =     DIX [AR2,P#6.1];
      L     #PVAct;
      T     DID [AR2,P#8.0];
      L     #State;
      T     DIW [AR2,P#48.0];	// #Objektstatus  (Struktur) 
END_FUNCTION

FUNCTION FC 30 : VOID
TITLE = Baustein vorbelegen
//Erstellung:
//Datum        Bearbeiter                                                 Version
//--------------------------------------------------------------------------------
//08.12.98     R.Schaffert (sra)                                          01.00.00
//
//Änderungen:
//Nr. Datum    Bearb Beschreibung                                   Marke Version
//--------------------------------------------------------------------------------
//01  13.04.00 sra   Fehlerbehebung (1 Byte zuviel belegt)                01.00.01
//02  25.08.00 sra   Fehlerbehebung Zeigerberechnung                      01.00.02
//
//________________________________________________________________________________
//Beschreibung:
//
//Diese Funktion beschreibt die angegebenen Worte eines Datenbausteins mit dem im 
//Parameter "Wert" eingetragenen Wert.
//
AUTHOR : sra
FAMILY : AZO
VERSION : 0.0
VAR_INPUT
  DB_Nr : INT ;	//Datenbausteinnummer
  DW_Anfang : INT ;	//Anfangs-Datenwort im Datenbaustein
  Anzahl_Bytes : INT ;	//Anzahl der Bytes die vorbelegt werden sollen
  Wert : INT ;	//Wert mit dem der Bereich vorbelegt werden soll
END_VAR
VAR_TEMP
  Datenbaustein : INT ;
  Ptr_aktuelles_Datenbyte : DWORD ;
  Ptr_Ende_Datenbyte : DWORD ;
END_VAR
BEGIN
NETWORK
TITLE = Anzahl Worte prüfen
      L     #Anzahl_Bytes;
      L     0;
      <=I;
      JC    Ende;
NETWORK
TITLE = Datenbaustein öffnen
      L     #DB_Nr;
      T     #Datenbaustein;
      OPN   DB [#Datenbaustein];
NETWORK
TITLE = Pointer belegen
      L     #DW_Anfang;
      SLD   3;
      T     #Ptr_aktuelles_Datenbyte;
      L     #Anzahl_Bytes;
      L     #DW_Anfang;
      +I;
      SLD   3;
      T     #Ptr_Ende_Datenbyte;
NETWORK
TITLE = Wert schreiben
Loop: NOP   0;
      L     #Wert;
      T     DBB [#Ptr_aktuelles_Datenbyte];
      L     #Ptr_aktuelles_Datenbyte;	// Wortadresse um 1 erhöhen
      L     P#1.0;
      +D;
      T     #Ptr_aktuelles_Datenbyte;
      L     #Ptr_Ende_Datenbyte;
      <D;
      JC    Loop;
Ende: NOP   0;
END_FUNCTION

FUNCTION FC 40 : VOID
TITLE = SST an Slave
//Erstellung:
//Datum        Bearbeiter                                                 Version
//--------------------------------------------------------------------------------
//22.03.01     R.Schaffert (sra)                                          01.00.00
//
//Änderungen:
//Nr. Datum    Bearb Beschreibung                                   Marke Version
//--------------------------------------------------------------------------------
//01  16.08.01 sra   Fehlerbeseitigung  Daten löschen               (001) 01.00.01
//02  31.08.01 sra   Daten von Ziel auch löschen wenn Ziel-DB 0 ist (002) 01.00.02
//
//________________________________________________________________________________
//Beschreibung: 
//
//Der Baustein kopiert die Schnittstelle, die durch den ANY-Zeiger festgelegt 
//ist, 
//an einen "Slave". Sobald ein Bit in der Steuerbitleiste gesetzt ist reagiert 
//der 
//Slave und antwortet. Ist kein Bit in der Steuerbitleiste belegt, baut der Slave 
//die Schnittstelle ab und kann durch anderen Master belegt werden.
//!!Die Steuerbitleiste ist immer das letzte Wort in der Schnittstelle!!
//
//Anwendung z.B. bei Kommunikation mehrere Waage <-> mehrere Silo  
// 
//
AUTHOR : sra
FAMILY : AZO
VERSION : 0.0
VAR_INPUT
  i_Freigabe : BOOL ;	//Freigabe der Kopierfunktion
  i_Ziel_DB : INT ;	//Ziel-Datenbaustein
  i_Ziel_DW : INT ;	//Ziel-Datenwort im Ziel-Datenbaustein
  i_SST_von_Ziel : ANY ;	//ANY-Zeiger auf Schnittstellen von Slave
  i_SST_an_Ziel : ANY ;	//ANY-Zeiger auf Schnittstellen an Slave
END_VAR
VAR_OUTPUT
  Ziel_frei : BOOL ;	//"Slave" ist nicht durch anderen Master belegt,die Daten können umkopiert werden
END_VAR
VAR_TEMP
  Quell_DB : INT ;
  SST_an_Anfangs_DW : INT ;
  SST_an_Laenge : INT ;
  SST_von_Anfangs_DW : INT ;
  SST_von_Laenge : INT ;
  Ziel_DB : INT ;
  Zaehler : INT ;
  Fehler_Blockkopieren : INT ;
END_VAR
BEGIN
NETWORK
TITLE = ANY Zeiger "SST_von_Ziel" zerlegen
      L     P##i_SST_von_Ziel;
      LAR2;
      L     W [AR2,P#2.0];
      T     #SST_von_Laenge;
      L     D [AR2,P#6.0];
      L     DW#16#FFFFFF;
      AD;
      SRD   3;
      T     #SST_von_Anfangs_DW;
NETWORK
TITLE = ANY Zeiger "SST_an_Ziel" zerlegen
      L     P##i_SST_an_Ziel;
      LAR2;
      L     W [AR2,P#2.0];
      T     #SST_an_Laenge;
      L     W [AR2,P#4.0];
      T     #Quell_DB;
      L     D [AR2,P#6.0];
      L     DW#16#FFFFFF;
      AD;
      SRD   3;
      T     #SST_an_Anfangs_DW;
NETWORK
TITLE = Prüfen ob Ziel-DB <> 0
      L     #i_Ziel_DB;
      L     0;
      ==I;
      JC    DEL1;	// 002
NETWORK
TITLE = Prüfen ob Slave belegt ist
      L     #i_Ziel_DB;
      T     #Ziel_DB;
      OPN   DB [#Ziel_DB];
      L     #i_Ziel_DW;
      SLD   3;
      LAR2;
      O(;	// Slave bereits belegt ?
      L     DBW [AR2,P#0.0];
      L     #Quell_DB;
      ==I;
      );
      O(;	// Slave frei ?
      L     DBW [AR2,P#0.0];
      L     0;
      ==I;
      );
      =     #Ziel_frei;
NETWORK
TITLE = Daten von Ziel löschen
DEL1: OPN   DB [#Quell_DB];
      L     #SST_von_Anfangs_DW;
      SLD   3;
      LAR2;
      L     #SST_von_Laenge;
DEL2: T     #Zaehler;
      L     0;
      T     DBB [AR2,P#0.0];
      L     P#1.0;	// (001)
      +AR2;	// (001)
      L     #Zaehler;
      LOOP  DEL2;
      ON    #i_Freigabe;
      ON    #Ziel_frei;
      O(;	// (002)
      L     #i_Ziel_DB;	// (002)
      L     0;	// (002)
      ==I;	// (002)
      );	// (002)
      BEC;
NETWORK
TITLE = Daten an Slave kopieren
      L     #SST_an_Anfangs_DW;
      SLD   3;
      LAR2;
      L     #Quell_DB;
      T     DBW [AR2,P#0.0];
      L     #SST_von_Anfangs_DW;
      T     DBW [AR2,P#2.0];
      CALL  FC 5 (
           Quell_Typ                := B#16#44,
           Quell_DB                 := #Quell_DB,
           Quell_DW                 := #SST_an_Anfangs_DW,
           Ziel_Typ                 := B#16#44,
           Ziel_DB                  := #i_Ziel_DB,
           Ziel_DW                  := #i_Ziel_DW,
           Block_Laenge             := #SST_an_Laenge,
           outFehler                := #Fehler_Blockkopieren);
END_FUNCTION

FUNCTION FC 41 : VOID
TITLE = SST an Master
//Erstellung:
//Datum        Bearbeiter                                                 Version
//--------------------------------------------------------------------------------
//22.03.01     R.Schaffert (sra)                                          01.00.00
//
//Änderungen:
//Nr. Datum    Bearb Beschreibung                                   Marke Version
//--------------------------------------------------------------------------------
//01  00.00.00 xxx   xxx                                            ???   01.xx.xx
//
//________________________________________________________________________________
//Beschreibung: 
//
//Der Baustein kopiert die Schnittstelle, die durch den ANY-Zeiger festgelegt 
//ist, an einen "Master". Sobald ein Bit in der Steuerbitleiste gesetzt ist 
//reagiert der Slave und antwortet. Ist kein Bit in der Steuerbitleiste belegt, 
//baut der Slave die Schnittstelle ab und kann durch anderen Master belegt werden.
//!!Die Steuerbitleiste ist immer das letzte Wort in der Schnittstelle!!
//
//Anwendung z.B. bei Kommunikation mehrere Waage <-> mehrere Silo  
// 
//
//
AUTHOR : sra
FAMILY : AZO
VERSION : 0.0
VAR_INPUT
  i_SST_von_Ziel : ANY ;	//ANY-Zeiger auf Schnittstelle von Master
  i_SST_an_Ziel : ANY ;	//ANY-Zeiger auf Schnittstelle an Master
END_VAR
VAR_TEMP
  SST_an_Anfangs_DW : INT ;
  SST_an_Laenge : INT ;
  SST_von_Anfangs_DW : INT ;
  SST_von_Laenge : INT ;
  Ptr_SST_von_Anfangs_DW : DWORD ;
  Ptr_SST_von_Steuerbits : DWORD ;	//Steuerbits = Anfangs-DW + Länge -2
  Quell_DB : INT ;
  Ziel_DB : INT ;
  Ziel_DW : INT ;
  Fehler_Blockkopieren : INT ;
END_VAR
BEGIN
NETWORK
TITLE = ANY Zeiger "SST_von_Ziel" zerlegen
      L     P##i_SST_von_Ziel;
      LAR2;
      L     W [AR2,P#2.0];	// Länge der Struktur
      T     #SST_von_Laenge;
      L     D [AR2,P#6.0];	// Anfangs-DW der Struktur
      L     DW#16#FFFFFF;
      AD;
      SRD   3;
      T     #SST_von_Anfangs_DW;
NETWORK
TITLE = ANY Zeiger "SST_an_Ziel" zerlegen
      L     P##i_SST_an_Ziel;
      LAR2;
      L     W [AR2,P#2.0];
      T     #SST_an_Laenge;
      L     W [AR2,P#4.0];
      T     #Quell_DB;
      L     D [AR2,P#6.0];
      L     DW#16#FFFFFF;
      AD;
      SRD   3;
      T     #SST_an_Anfangs_DW;
NETWORK
TITLE = Pointer bilden
      L     #SST_von_Anfangs_DW;
      SLD   3;
      T     #Ptr_SST_von_Anfangs_DW;
      L     #SST_von_Anfangs_DW;
      L     #SST_von_Laenge;
      +I;
      L     2;
      -I;
      SLD   3;
      T     #Ptr_SST_von_Steuerbits;
NETWORK
TITLE = Prüfen ob Anforderung vorhanden
      OPN   DB [#Quell_DB];
      O(;
      L     DBW [#Ptr_SST_von_Anfangs_DW];	// Ziel-DB
      L     0;
      ==I;
      );
      O(;
      L     DBW [#Ptr_SST_von_Steuerbits];	// Steuerbits
      L     0;
      ==I;
      );
      JC    DEL;
NETWORK
TITLE = Daten an Master kopieren
      LAR2  #Ptr_SST_von_Anfangs_DW;
      L     DBW [AR2,P#0.0];	// Ziel-DB aus Struktur "SST_von" ermitteln
      T     #Ziel_DB;
      L     DBW [AR2,P#2.0];	// Ziel-DW aus Struktur "SST_von" ermitteln
      T     #Ziel_DW;
      CALL  FC 5 (
           Quell_Typ                := B#16#44,
           Quell_DB                 := #Quell_DB,
           Quell_DW                 := #SST_an_Anfangs_DW,
           Ziel_Typ                 := B#16#44,
           Ziel_DB                  := #Ziel_DB,
           Ziel_DW                  := #Ziel_DW,
           Block_Laenge             := #SST_an_Laenge,
           outFehler                := #Fehler_Blockkopieren);
NETWORK
TITLE = Daten von Master löschen
DEL:  L     DBW [#Ptr_SST_von_Steuerbits];
      L     0;
      <>I;
      JC    DELS;
      L     0;
      T     DBW [#Ptr_SST_von_Anfangs_DW];
DELS: L     0;
      T     DBW [#Ptr_SST_von_Steuerbits];
END_FUNCTION

FUNCTION FC 47 : VOID
TITLE = Tabelle schreiben
//DATUM     BEARBEITER                                                    VERSION
//--------------------------------------------------------------------------------
//29.02.00  A. Geiger (gea)                                               01.00.00
//  
//Änderungen:
//Nr. Datum    Bearb Beschreibung                                   Marke Version
//--------------------------------------------------------------------------------
//01  30.08.00 gea   Neue Konzeption (Kopieren über Schleife)             02.00.00
//
//________________________________________________________________________________
//Beschreibung: 
//Datensatz in Tabelle schreiben
//
//Aufbau Tabelle:
//  Tabellen-DB: 
//               DBB0    ... DBB(n-1)  1.Zeile
//               DBB(n)  ... DBB(2n-1) 2.Zeile
//               DBB(2n) ... DBB(3n-1) 3.Zeile
//               usw.
//
//Die Anzahl der Spalten pro Zeile (n) ist abhängig von der Länge der "Quelle".
//Die "Quelle" muß ein ANY-Zeiger auf Bytes oder Stuct sein.
//eine Überprüfung auf Existenz und Länge des Tabellen-DBs wird durchgeführt.
//
AUTHOR : gea
FAMILY : AZO
VERSION : 0.0
VAR_INPUT
  in_Tabelle_DB : INT ;	//Tabellen-DB-Nr.
  in_Offset_DW : INT ;	//Offset erster Tabelleneintrag in Tabellen-DB
  in_Zeile_schreiben : INT ;	//Eintrag in Tabelle, der geschrieben werden soll
END_VAR
VAR_OUTPUT
  out_Fehler : INT ;	//Fehlerauswertung
END_VAR
VAR_IN_OUT
  io_Quelle : ANY ;	//Zeiger auf Quelldaten Block
END_VAR
VAR_TEMP
  G_DB_SAVE : INT ;	//Global-DB-Register
  I_DB_SAVE : INT ;	//Instanz-DB-Register
  Zeiger_Quelle : DWORD ;
  DB_Quelle : INT ;
  Zeiger_Ziel : DWORD ;
  DB_Ziel : INT ;
  Blocklaenge : INT ;
  Datentyp : BYTE ;
  Start_DBB : INT ;
END_VAR
BEGIN
NETWORK
TITLE = DB-Register sichern
      L     DBNO;
      T     #G_DB_SAVE;
      L     DINO;
      T     #I_DB_SAVE;
NETWORK
TITLE = ANY-Zeiger Quelle zerlegen
      L     P##io_Quelle;
      LAR1;
      L     B [AR1,P#1.0];
      T     #Datentyp;
      L     W [AR1,P#2.0];
      T     #Blocklaenge;
      L     W [AR1,P#4.0];
      T     #DB_Quelle;
      L     D [AR1,P#6.0];
      T     #Zeiger_Quelle;
NETWORK
TITLE = Blocklänge prüfen
      L     #Blocklaenge;
      L     0;
      <=I;
      JC    BLFE;	//Blocklänge Fehler
NETWORK
TITLE = Datentyp prüfen
      L     #Datentyp;
      L     2;	//Datentyp = Byte oder Struct
      ==I;
      JCN   DTFE;
NETWORK
TITLE = Start-DBB des gewählten Eintrags
      L     #in_Zeile_schreiben;
      L     1;
      -I;
      L     #Blocklaenge;
      *I;
      L     #in_Offset_DW;
      +I;
      T     #Start_DBB;	//Start des n-ten Eintrags
NETWORK
TITLE = Bereichszeiger Zielzeiger
      L     W#16#85;
      CAD;
      L     #Start_DBB;
      SLD   3;
      +D;
      T     #Zeiger_Ziel;
NETWORK
TITLE = Ziel-DB
      L     #in_Tabelle_DB;
      T     #DB_Ziel;
NETWORK
TITLE = DBs aufschlagen
      L     #DB_Quelle;
      L     0;
      <>I;
      JCN   QNDB;
      OPN   DB [#DB_Quelle];
      L     DBNO;
      L     0;
      <=I;
      JC    DBNX;	//Fehler DB existiert nicht
      L     #Zeiger_Quelle;
      SRW   3;	//Anfangsbyte
      L     #Blocklaenge;
      +I;
      L     DBLG;
      >I;
      JC    DBLF;	//Fehler DB Länge nicht ausreichend
      L     #Zeiger_Quelle;
      L     DW#16#FFFFFF;
      AD;
      L     W#16#84;
      CAD;
      +D;
      T     #Zeiger_Quelle;
QNDB: L     #DB_Ziel;
      L     0;
      <>I;
      JCN   ZNDB;
      OPN   DI [#DB_Ziel];
      L     DINO;
      L     0;
      <=I;
      JC    DBNX;	//Fehler DB existiert nicht
      L     #Start_DBB;
      L     #Blocklaenge;
      +I;
      L     DILG;
      >I;
      JC    DBLF;	//Fehler DB Länge nicht ausreichend
ZNDB: NOP   0;
NETWORK
TITLE = Bytes kopieren
//geschwindigkeitsopitmiert:
//- Schleifenzäehler bleibt in AKKU1 und AKKU2
//- Kopieren über Worte, letztes Byte (ungerade Bytezahl) separat.
// (network holds code this reader does not know; not shown)
NETWORK
TITLE = Fehlerauswertung
      L     0;	//kein Fehler
      JU    SEFE;	//  setze Fehlerausgang
      L     -1;	//Bereichszeiger Quelle falsch
      JU    SEFE;	//  setze Fehlerausgang
      L     -2;	//Bereichszeiger Ziel falsch
      JU    SEFE;	//  setze Fehlerausgang
BLFE: L     -3;	//Blocklänge falsch
      JU    SEFE;	//  setze Fehlerausgang
DBNX: L     -4;	//Datenbaustein nicht existent 
      JU    SEFE;	//  setze Fehlerausgang
DBLF: L     -5;	//Datenbaustein Längenfehler
      JU    SEFE;	//  setze Fehlerausgang
DTFE: L     -6;	//Fehler Datentyp in ANY-Zeiger
SEFE: T     #out_Fehler;
NETWORK
TITLE = DB-Register wiederherstellen
      OPN   DB [#G_DB_SAVE];
      OPN   DI [#I_DB_SAVE];
NETWORK
TITLE = BIE-Bit zuweisen
      L     #out_Fehler;
      L     0;
      ==I;
      SAVE;
END_FUNCTION

FUNCTION FC 104 : VOID
TITLE = BlockTransfer mit ANY-Zeiger als Ziel
//DATUM     BEARBEITER                                                    VERSION
//--------------------------------------------------------------------------------
//29.02.00  A. Geiger (gea)                                               01.00.00
//  
//Änderungen:
//Nr. Datum    Bearb Beschreibung                    Änderung       Marke Version
//--------------------------------------------------------------------------------
//01  06.07.00 gea   Neue Konzeption (Kopieren über Schleife)             02.00.00
//02  26.10.01 gea   Fehlerbehebung DB überprüfen                   (002) 02.00.01
//03  05.11.03 gea   Alle Datentypen zulassen                       (003) 02.00.02
//04  10.06.10 sra   Bereich > 32767 kopieren                       (004) 02.00.03
//________________________________________________________________________________
//
//Funktion:
//
//Beschreibung: Kopieren Quelle nach Ziel (ANY-Zeiger)
//
//Datentyp:
//  P - Peripherie
//  E - Eingänge
//  A - Ausgänge
//  M - Merker
//  D - Datenbaustein in Quell_DB bzw. Ziel_DB
//  I - Instanz-DB in DI-Register
//  G - Global-DB in DB-Register
//  L - Lokaldaten
//  K - Bausteinvorbelegen mit Konstante in Quell_DW (Low-Byte) (nur für Quelle)
//
//
//
//
//
//
//
//
//
//
//
//
//
//THE HORROR CONTINUES ...
AUTHOR : gea
VERSION : 0.0
VAR_INPUT
  in_Quell_Typ : CHAR ;
  in_Quell_DB : INT ;	//Ziel-DB bei DW-Transfer
  in_Quell_DW : INT ;	//Byte-Adresse der Quelle
  in_Ziel : ANY ;
END_VAR
VAR_OUTPUT
  out_Fehler : INT ;	//Fehlermeldung
END_VAR
VAR_TEMP
  G_DB_SAVE : INT ;	//Global-DB-Register
  I_DB_SAVE : INT ;	//Instanz-DB-Register
  Zeiger_Quelle : DWORD ;
  DB_Quelle : INT ;
  Zeiger_Ziel : DWORD ;
  DB_Ziel : INT ;
  Blocklaenge : INT ;
  Datentyp : BYTE ;
END_VAR
BEGIN
NETWORK
TITLE = DB-Register sichern
      L     DBNO;
      T     #G_DB_SAVE;
      L     DINO;
      T     #I_DB_SAVE;
NETWORK
TITLE = ANY-Zeiger Ziel zerlegen
      L     P##in_Ziel;
      LAR1;
      L     B [AR1,P#1.0];
      T     #Datentyp;
      L     W [AR1,P#2.0];
      T     #Blocklaenge;
      L     W [AR1,P#4.0];
      T     #DB_Ziel;
      L     D [AR1,P#6.0];
      T     #Zeiger_Ziel;
NETWORK
TITLE = Blocklänge prüfen
      L     #Blocklaenge;
      L     0;
      <=I;
      JC    BLFE;	//Blocklänge Fehler
NETWORK
TITLE = Datentyp prüfen
      L     #Datentyp;
      L     0;	//Datentyp = Byte oder Struct //(003)
      <>I;
      JCN   DTFE;
NETWORK
TITLE = Bereichskennung Quellzeiger
      L     #in_Quell_Typ;
      L     'P';
      ==I;
      L     W#16#80;
      JC    BEKQ;
      L     #in_Quell_Typ;
      L     'E';
      ==I;
      L     W#16#81;
      JC    BEKQ;
      L     #in_Quell_Typ;
      L     'A';
      ==I;
      L     W#16#82;
      JC    BEKQ;
      L     #in_Quell_Typ;
      L     'M';
      ==I;
      L     W#16#83;
      JC    BEKQ;
      L     #in_Quell_Typ;
      L     'D';
      ==I;
      L     W#16#84;
      JC    BEKQ;
      L     #in_Quell_Typ;
      L     'I';
      ==I;
      L     W#16#84;
      JC    BEKQ;
      L     #in_Quell_Typ;
      L     'G';
      ==I;
      L     W#16#84;
      JC    BEKQ;
      L     #in_Quell_Typ;
      L     'L';
      ==I;
      L     W#16#87;
      JC    BEKQ;
      L     #in_Quell_Typ;
      L     'K';
      ==I;
      L     L#0;
      JC    BEK1;
      JU    BEFQ;	//Bereichskennung falsch Quelle
BEKQ: CAD;
      L     #in_Quell_DW;
      SLD   3;
      +D;
BEK1: T     #Zeiger_Quelle;
NETWORK
TITLE = Quell-DB
      L     #in_Quell_Typ;
      L     'D';
      ==I;
      L     #in_Quell_DB;
      JC    DBQ;
      L     #in_Quell_Typ;
      L     'I';
      ==I;
      L     DINO;
      JC    DBQ;
      L     #in_Quell_Typ;
      L     'G';
      ==I;
      L     DBNO;
      JC    DBQ;
      L     0;
DBQ:  T     #DB_Quelle;
NETWORK
TITLE = DBs aufschlagen
      O(;	//(002)
      L     #in_Quell_Typ;	//(002)
      L     'D';	//(002)
      ==I;	//(002)
      );	//(002)
      O(;	//(002)
      L     #in_Quell_Typ;	//(002)
      L     'I';	//(002)
      ==I;	//(002)
      );	//(002)
      O(;	//(002)
      L     #in_Quell_Typ;	//(002)
      L     'G';	//(002)
      ==I;	//(002)
      );	//(002)
      JCN   QNDB;
      OPN   DB [#DB_Quelle];
      L     DBNO;
      L     0;
      <=I;
      JC    DBNX;	//Fehler DB existiert nicht
      L     #in_Quell_DW;
      L     #Blocklaenge;
      +D;	// (004)
      L     DBLG;
      >D;	// (004)
      JC    DBLF;	//Fehler DB Länge nicht ausreichend
QNDB: L     #DB_Ziel;
      L     0;
      <>I;
      JCN   ZNDB;
      OPN   DI [#DB_Ziel];
      L     DINO;
      L     0;
      <=I;
      JC    DBNX;	//Fehler DB existiert nicht
      L     #Zeiger_Ziel;
      SRW   3;	//Anfangsbyte
      L     #Blocklaenge;
      +D;	// (004)
      L     DILG;
      >D;	// (004)
      JC    DBLF;	//Fehler DB Länge nicht ausreichend
      L     #Zeiger_Ziel;
      L     DW#16#FFFFFF;
      AD;
      L     W#16#85;
      CAD;
      +D;
      T     #Zeiger_Ziel;
ZNDB: NOP   0;
NETWORK
TITLE = Bereich vorbelegen
//geschwindigkeitsopitmiert:
//- Schleifenzäehler bleibt in AKKU1 und AKKU2
//- Kopieren über Worte, letztes Byte (ungerade Bytezahl) separat.
      L     #in_Quell_Typ;
      L     'K';
      ==I;
      JCN   NKCO;
      L     #Zeiger_Ziel;
      LAR2;
      L     #in_Quell_DW;	//Konstante für vorbelegen
      L     #in_Quell_DW;
      SLW   8;	//  In AKKU1LL und AKKU1LH
      OW;
      L     #Blocklaenge;	//Schleifenzähler Blocklaenge->AKKU1
      SRW   1;
SCHK: TAK;	//Schleifenzähler AKKU1->AKKU2; Vorbelegwert in AKKU1
      T     W [AR2,P#0.0];
      +AR2  P#2.0;
      TAK;	//Schleifenzähler in AKKU2->AKKU1; Vorbelegwert in AKKU2
      LOOP  SCHK;
      JZ    BLGK;	//Gerade Byteanzahl A1=0 und A0=0 nach "SRW 1"
      L     #in_Quell_DW;	//Ungerade Bytezahl letztes Byte einzeln Kopieren
      SRW   8;
      T     B [AR2,P#0.0];
BLGK: NOP   0;
      JU    BLGE;
NKCO: NOP   0;
NETWORK
TITLE = Bytes kopieren
//geschwindigkeitsopitmiert:
//- Schleifenzäehler bleibt in AKKU1 und AKKU2
//- Kopieren über Worte, letztes Byte (ungerade Bytezahl) separat.
// (network holds code this reader does not know; not shown)
NETWORK
TITLE = Fehlerauswertung
      L     0;	//kein Fehler
      JU    SEFE;	//  setze Fehlerausgang
BEFQ: L     -1;	//Bereichszeiger Quelle falsch
      JU    SEFE;	//  setze Fehlerausgang
      L     -2;	//Bereichszeiger Ziel falsch
      JU    SEFE;	//  setze Fehlerausgang
BLFE: L     -3;	//Blocklänge falsch
      JU    SEFE;	//  setze Fehlerausgang
DBNX: L     -4;	//Datenbaustein nicht existent 
      JU    SEFE;	//  setze Fehlerausgang
DBLF: L     -5;	//Datenbaustein Längenfehler
      JU    SEFE;	//  setze Fehlerausgang
DTFE: L     -6;	//Fehler Datentyp in ANY-Zeiger
SEFE: T     #out_Fehler;
NETWORK
TITLE = DB-Register wiederherstellen
      OPN   DB [#G_DB_SAVE];
      OPN   DI [#I_DB_SAVE];
NETWORK
TITLE = BIE-Bit zuweisen
      L     #out_Fehler;
      L     0;
      ==I;
      SAVE;
END_FUNCTION

FUNCTION FC 113 : VOID
TITLE = function for several cabinets with their own fuse check
//Erstellung:
//Date        developer                                                  version
//--------------------------------------------------------------------------------
//18.07.2016  A.Kremer (kal)                                             01.00.00
//
//changes:
//No. Date    developer description                                 Mark  version
//--------------------------------------------------------------------------------
//
//________________________________________________________________________________
//function:
//function, if more than one cabinet handle their own fuse check.
//function can be called several times, then.
//
AUTHOR : kal
FAMILY : AZO
VERSION : 0.0
VAR_INPUT
  iFaultFuse_OK : BOOL ;	//Eingang Sicherung OK = Eingang Störung Sicherung
END_VAR
VAR_OUTPUT
  qlFaultFuse : BOOL ;	//Ausgang der Lampe "Störung Sicherung"
  qFaultFuse : BOOL ;	//Störung Sicherung -> für Störbitzuweisung im DB34
END_VAR
BEGIN
NETWORK
TITLE = lamp "fault fuse" and fault message
      AN    #iFaultFuse_OK;
      =     #qlFaultFuse;
      =     #qFaultFuse;
END_FUNCTION

FUNCTION FC 6079 : INT
TITLE = simulate analog signal
//creation:
//date         who                                                         version
//--------------------------------------------------------------------------------
//28.12.2010   M. Junker (jm)                                             01.00.00
//
//changes:
//no. date       who            what                                       version
//--------------------------------------------------------------------------------
// 1  
//
//Function:
//simulates a slow changing analog signal (pressure, temperature) for 
//visualization tests or program tests
//
//y = a * sin(x) + b
AUTHOR : jm
FAMILY : AZO
NAME : SIMUL
VERSION : 0.1
VAR_INPUT
  RELEASE : BOOL ;	//release simulation
  PERIOD : REAL ;	//period time for sin() [s]
  MAX : REAL ;	//maximum analog value to simulate
  MIN : REAL ;	//minimum analog value to simulate
  DEFAULT : REAL ;	//default value if not simulating
  MAXVALUE : REAL ;	//upper limit analog value
  MINVALUE : REAL ;	//lower limit analog value
END_VAR
VAR_OUTPUT
  RET_VAL : INT ;	//simulated analog signal
END_VAR
VAR_IN_OUT
  STARTTIME : TIME ;	//starttime [ms]
  ONESHOTSTART : BOOL ;	//help flag start
END_VAR
VAR_TEMP
  ACTTIME : TIME ;
  y : REAL ;
  x : REAL ;
  a : REAL ;
  b : REAL ;
  MR1 : REAL ;
  MR2 : REAL ;
END_VAR
BEGIN
NETWORK
TITLE = detect start time
      A     #RELEASE;
      FP    #ONESHOTSTART;
      JCN   NSST;	// Not Set Start Time
      CALL  SFC 64 (
           RET_VAL                  := #STARTTIME);
NSST: NOP   0;
NETWORK
TITLE = check if simulation necessary
      A     #RELEASE;
      JC    CONT;
      L     #DEFAULT;
      T     #y;
      JU    OUT;	// scale value for output
NETWORK
TITLE = calculate x
//x = 2*pi/1000/PERIOD*deltaTms = deltaTms*pi/500/PERIOD
CONT: CALL  SFC 64 (
           RET_VAL                  := #ACTTIME);
      L     #ACTTIME;
      L     #STARTTIME;
      -D;	// deltaT in ms 
      DTR;
      L     3.141593e+00;	// PI
      *R;
      L     5.000000e+02;
      /R;
      L     #PERIOD;
      /R;
      T     #x;
NETWORK
TITLE = calculate a
//a = (MAX-MIN)/2
      L     #MAX;
      L     #MIN;
      -R;
      L     2.000000e+00;
      /R;
      T     #a;
NETWORK
TITLE = calculate b
//b = (MAX+MIN)/2
      L     #MAX;
      L     #MIN;
      +R;
      L     2.000000e+00;
      /R;
      T     #b;
NETWORK
TITLE = calculate y
//y = a*sin(x)+b
// (network holds code this reader does not know; not shown)
NETWORK
TITLE = scale output
//z = (MAXDIGIT-MINDIGIT)/(MAXVALUE-MINVALUE)*(y-MINVALUE)+MINDIGIT 
OUT:  L     #MAXVALUE;
      L     #MINVALUE;
      -R;
      T     #MR1;
      L     #y;
      L     #MINVALUE;
      -R;
      T     #MR2;
      L     2.764800e+04;
      L     #MR1;
      /R;
      L     #MR2;
      *R;
      RND;
      T     #RET_VAL;
END_FUNCTION

FUNCTION FC 6091 : VOID
TITLE = simulate valve 3A3E
//creation:
//date         who                                                         version
//--------------------------------------------------------------------------------
//04.12.2015   M. Junker (jm)                                             01.00.00
//
//changes:
//no. date       who            what                                       version
//--------------------------------------------------------------------------------
// 1  
//
//Function:
//simulate valve
AUTHOR : jm
FAMILY : AZO
NAME : SIMUL
VERSION : 1.0
VAR_INPUT
  o_ValveOn : BOOL ;
  o_ValveOff : BOOL ;
  o_ValveSealup : BOOL ;
END_VAR
VAR_OUTPUT
  i_ValveOn : BOOL ;	//on, open, pos1, ...
  i_ValveOff : BOOL ;	//off, closed, pos2, ...
  i_ValveSealed : BOOL ;	//sealed
END_VAR
VAR_IN_OUT
  mPosition : BOOL ;	//help memory
END_VAR
BEGIN
NETWORK
TITLE = valve on
      A     #o_ValveOn;
      S     #mPosition;
NETWORK
TITLE = valve off
      A     #o_ValveOff;
      R     #mPosition;
NETWORK
TITLE = indications
      A     #mPosition;
      =     #i_ValveOn;
      NOT;
      =     #i_ValveOff;
NETWORK
TITLE = sealed
      A     #o_ValveSealup;
      =     #i_ValveSealed;
END_FUNCTION

FUNCTION FC 6092 : VOID
TITLE = simulate valve 2A2E (dosing valve)
//creation:
//date         who                                                         version
//--------------------------------------------------------------------------------
//05.06.2014   M. Junker (jm)                                             01.00.00
//
//changes:
//no. date       who            what                                       version
//--------------------------------------------------------------------------------
// 1  
//
//Function:
//simulate valve
AUTHOR : jm
FAMILY : AZO
NAME : SIMUL
VERSION : 1.0
VAR_INPUT
  in_Ventil_Typ : INT ;	//siehe Funktionsbeschreibung unten
  o_ValveCoarse : BOOL ;
  o_ValveFine : BOOL ;
END_VAR
VAR_OUTPUT
  i_ValveOpen : BOOL ;	//on, open, pos1, ...
  i_ValveClosed : BOOL ;	//off, closed, pos2, ...
END_VAR
VAR_IN_OUT
  mPosition : BOOL ;	//help memory
END_VAR
BEGIN
NETWORK
TITLE = valve open
      A     #o_ValveCoarse;
      S     #mPosition;
NETWORK
TITLE = valve  closed
      AN    #o_ValveCoarse;
      AN    #o_ValveFine;
      R     #mPosition;
NETWORK
TITLE = valve type 0
      A(;
      L     #in_Ventil_Typ;
      L     0;
      );
      <>I;
      JC    NVT0;
      A     #o_ValveCoarse;
      =     #i_ValveOpen;
      AN    #o_ValveCoarse;
      AN    #o_ValveFine;
      =     #i_ValveClosed;
NVT0: NOP   0;
NETWORK
TITLE = valve type 1
      A(;
      L     #in_Ventil_Typ;
      L     1;
      );
      <>I;
      JC    NVT1;
      A     #mPosition;
      =     #i_ValveOpen;
      AN    #mPosition;
      =     #i_ValveClosed;
NVT1: NOP   0;
NETWORK
TITLE = valve type 2
      A(;
      L     #in_Ventil_Typ;
      L     2;
      );
      <>I;
      JC    NVT2;
      A     #mPosition;
      =     #i_ValveOpen;
      AN    #mPosition;
      =     #i_ValveClosed;
NVT2: NOP   0;
END_FUNCTION

FUNCTION FC 6093 : VOID
TITLE = simulate valve 2A2E (double seat)
//creation:
//date         who                                                         version
//--------------------------------------------------------------------------------
//27.05.2014   M. Junker (jm)                                             01.00.00
//
//changes:
//no. date       who            what                                       version
//--------------------------------------------------------------------------------
// 1  
//
//Function:
//simulate valve
AUTHOR : jm
FAMILY : AZO
NAME : SIMUL
VERSION : 1.0
VAR_INPUT
  o_Valve_E0 : BOOL ;
  o_Valve_E1 : BOOL ;
END_VAR
VAR_OUTPUT
  i_Valve_A0 : BOOL ;	//on, open, pos1, ...
  i_Valve_A1 : BOOL ;	//off, closed, pos2, ...
END_VAR
BEGIN
NETWORK
TITLE = valve open
      A     #o_Valve_E0;
      A     #o_Valve_E1;
      =     #i_Valve_A1;
NETWORK
TITLE = valve close
      ON    #o_Valve_E0;
      ON    #o_Valve_E1;
      =     #i_Valve_A0;
END_FUNCTION

FUNCTION FC 6094 : VOID
TITLE = simulate motor 2A2E+iso
//creation:
//date         who                                                         version
//--------------------------------------------------------------------------------
//05.06.2014   M. Junker (jm)                                             01.00.00
//
//changes:
//no. date       who            what                                       version
//--------------------------------------------------------------------------------
// 1  
//
//Function:
//simulate motor + isolator
AUTHOR : jm
FAMILY : AZO
NAME : SIMUL
VERSION : 1.0
VAR_INPUT
  o_MotorCW : BOOL ;
  o_MotorACW : BOOL ;
  Isolators : BOOL ;
END_VAR
VAR_OUTPUT
  i_MotorCW : BOOL ;
  i_MotorACW : BOOL ;
  i_IsoMotor : BOOL ;
END_VAR
BEGIN
NETWORK
TITLE = motor CW
      A     #o_MotorCW;
      =     #i_MotorCW;
NETWORK
TITLE = motor ACW
      A     #o_MotorACW;
      =     #i_MotorACW;
NETWORK
TITLE = isolator
      A     #Isolators;
      =     #i_IsoMotor;
END_FUNCTION

FUNCTION FC 6095 : VOID
TITLE = simulate valve 2A2E
//creation:
//date         who                                                         version
//--------------------------------------------------------------------------------
//25.10.2010   M. Junker (jm)                                             01.00.00
//
//changes:
//no. date       who            what                                       version
//--------------------------------------------------------------------------------
// 1  
//
//Function:
//simulate valve
AUTHOR : jm
FAMILY : AZO
NAME : SIMUL
VERSION : 1.0
VAR_INPUT
  o_ValveOn : BOOL ;
  o_ValveOff : BOOL ;
END_VAR
VAR_OUTPUT
  i_ValveOn : BOOL ;	//on, open, pos1, ...
  i_ValveOff : BOOL ;	//off, closed, pos2, ...
END_VAR
VAR_IN_OUT
  mPosition : BOOL ;	//help memory
END_VAR
BEGIN
NETWORK
TITLE = valve on
      A     #o_ValveOn;
      S     #mPosition;
NETWORK
TITLE = valve off
      A     #o_ValveOff;
      R     #mPosition;
NETWORK
TITLE = indications
      A     #mPosition;
      =     #i_ValveOn;
      NOT;
      =     #i_ValveOff;
END_FUNCTION

FUNCTION FC 6096 : VOID
TITLE = simulate valve 1AE1
//creation:
//date         who                                                         version
//--------------------------------------------------------------------------------
//25.10.2010   M. Junker (jm)                                             01.00.00
//
//changes:
//no. date       who            what                                       version
//--------------------------------------------------------------------------------
// 1  
//
//Function:
//simulate valve
AUTHOR : jm
FAMILY : AZO
NAME : SIMUL
VERSION : 1.0
VAR_INPUT
  o_ValveOn : BOOL ;
END_VAR
VAR_OUTPUT
  i_ValveOff : BOOL ;	//off, closed, pos2, ...
END_VAR
BEGIN
NETWORK
TITLE = valve off
      AN    #o_ValveOn;
      =     #i_ValveOff;
END_FUNCTION

FUNCTION FC 6097 : VOID
TITLE = simulate valve 1A1E
//creation:
//date         who                                                         version
//--------------------------------------------------------------------------------
//25.10.2010   M. Junker (jm)                                             01.00.00
//
//changes:
//no. date       who            what                                       version
//--------------------------------------------------------------------------------
// 1  
//
//Function:
//simulate valve
AUTHOR : jm
FAMILY : AZO
NAME : SIMUL
VERSION : 1.0
VAR_INPUT
  o_ValveOn : BOOL ;
END_VAR
VAR_OUTPUT
  i_ValveOn : BOOL ;	//on, open, pos1, ...
END_VAR
BEGIN
NETWORK
TITLE = valve on
      A     #o_ValveOn;
      =     #i_ValveOn;
END_FUNCTION

FUNCTION FC 6098 : VOID
TITLE = simulate valve 1A2E
//creation:
//date         who                                                         version
//--------------------------------------------------------------------------------
//25.10.2010   M. Junker (jm)                                             01.00.00
//
//changes:
//no. date       who            what                                       version
//--------------------------------------------------------------------------------
// 1  
//
//Function:
//simulate valve
AUTHOR : jm
FAMILY : AZO
NAME : SIMUL
VERSION : 1.0
VAR_INPUT
  o_ValveOn : BOOL ;
END_VAR
VAR_OUTPUT
  i_ValveOn : BOOL ;	//on, open, pos1, ...
  i_ValveOff : BOOL ;	//off, closed, pos2, ...
END_VAR
BEGIN
NETWORK
TITLE = valve on
      A     #o_ValveOn;
      =     #i_ValveOn;
NETWORK
TITLE = valve off
      AN    #o_ValveOn;
      =     #i_ValveOff;
END_FUNCTION

FUNCTION FC 6099 : VOID
TITLE = simulate motor 1A1E+iso
//creation:
//date         who                                                         version
//--------------------------------------------------------------------------------
//25.10.2010   M. Junker (jm)                                             01.00.00
//
//changes:
//no. date       who            what                                       version
//--------------------------------------------------------------------------------
// 1  
//
//Function:
//simulate motor + isolator
AUTHOR : jm
FAMILY : AZO
NAME : SIMUL
VERSION : 1.0
VAR_INPUT
  o_MotorOn : BOOL ;
  Isolators : BOOL ;
END_VAR
VAR_OUTPUT
  i_MotorOn : BOOL ;
  i_IsoMotor : BOOL ;
END_VAR
BEGIN
NETWORK
TITLE = motor
      A     #o_MotorOn;
      =     #i_MotorOn;
NETWORK
TITLE = isolator
      A     #Isolators;
      =     #i_IsoMotor;
END_FUNCTION

DATA_BLOCK DB 2
VERSION : 0.0
FB 2
BEGIN
END_DATA_BLOCK

